LIN {X 0,Y 353.68,Z 667.866,A -85,B 0,C 180,E1 -13495.441,E2 -13495.441} C_VEL
LIN {X 0,Y 353.682,Z 668.66,A -85,B 0,C 180,E1 -13496.583,E2 -13496.583} C_VEL
LIN {X 0,Y 353.463,Z 669.191,A -85,B 0,C 180,E1 -13498.861,E2 -13498.861} C_VEL
LIN {X 0,Y 353.397,Z 668.253,A -85,B 0,C 180,E1 -13501.14,E2 -13501.14} C_VEL
LIN {X 0,Y 353.398,Z 665.846,A -85,B 0,C 180,E1 -13503.42,E2 -13503.42} C_VEL
LIN {X 0,Y 353.541,Z 663.076,A -85,B 0,C 180,E1 -13505.132,E2 -13505.132} C_VEL
LIN {X 0,Y 353.829,Z 657.939,A -85,B 0,C 180,E1 -13507.418,E2 -13507.418} C_VEL
LIN {X 0,Y 354.1,Z 652.954,A -85,B 0,C 180,E1 -13509.136,E2 -13509.136} C_VEL
LIN {X 0,Y 354.652,Z 645.736,A -85,B 0,C 180,E1 -13511.14,E2 -13511.14} C_VEL
LIN {X 0,Y 355.365,Z 638.179,A -85,B 0,C 180,E1 -13512.855,E2 -13512.855} C_VEL
LIN {X 0,Y 356.178,Z 628.788,A -85,B 0,C 180,E1 -13514.626,E2 -13514.626} C_VEL
LIN {X 0,Y 357.149,Z 618.14,A -85,B 0,C 180,E1 -13516.285,E2 -13516.285} C_VEL
LIN {X 0,Y 358.299,Z 605.968,A -85,B 0,C 180,E1 -13517.848,E2 -13517.848} C_VEL
LIN {X 0,Y 359.381,Z 593.917,A -85,B 0,C 180,E1 -13519.121,E2 -13519.121} C_VEL
LIN {X 0,Y 360.455,Z 580.861,A -85,B 0,C 180,E1 -13520.248,E2 -13520.248} C_VEL
LIN {X 0,Y 361.486,Z 566.317,A -85,B 0,C 180,E1 -13521.237,E2 -13521.237} C_VEL
LIN {X 0,Y 362.333,Z 551.357,A -85,B 0,C 180,E1 -13521.999,E2 -13521.999} C_VEL
LIN {X 0,Y 363.06,Z 535.678,A -85,B 0,C 180,E1 -13522.552,E2 -13522.552} C_VEL
LIN {X 0,Y 366.741,Z 431.293,A -85,B 0,C 180,E1 -13525.312,E2 -13525.312} C_VEL
LIN {X 0,Y 361.436,Z 398.032,A -85,B 0,C 180,E1 -13526.613,E2 -13526.613} C_VEL
LIN {X 0,Y 361.949,Z 391.941,A -85,B 0,C 180,E1 -13527.776,E2 -13527.776} C_VEL
LIN {X 0,Y 359.699,Z 381.366,A -85,B 0,C 180,E1 -13530.108,E2 -13530.108} C_VEL
LIN {X 0,Y 356.197,Z 366.492,A -85,B 0,C 180,E1 -13533.536,E2 -13533.536} C_VEL
LIN {X 0,Y 354.88,Z 361.062,A -85,B 0,C 180,E1 -13534.895,E2 -13534.895} C_VEL
LIN {X 0,Y 354.793,Z 360.917,A -85,B 0,C 180,E1 -13537.885,E2 -13537.885} C_VEL
LIN {X 0,Y 354.768,Z 360.912,A -85,B 0,C 180,E1 -13541.167,E2 -13541.167} C_VEL
LIN {X 0,Y 354.759,Z 360.919,A -85,B 0,C 180,E1 -13544.505,E2 -13544.505} C_VEL
LIN {X 0,Y 354.782,Z 360.903,A -85,B 0,C 180,E1 -13547.661,E2 -13547.661} C_VEL
LIN {X 0,Y 354.804,Z 361.09,A -85,B 0,C 180,E1 -13551.115,E2 -13551.115} C_VEL
LIN {X 0,Y 359.178,Z 374.687,A -85,B 0,C 180,E1 -13554.055,E2 -13554.055} C_VEL
LIN {X 0,Y 363.071,Z 388.801,A -85,B 0,C 180,E1 -13556.835,E2 -13556.835} C_VEL
LIN {X 0,Y 365.06,Z 396.769,A -85,B 0,C 180,E1 -13558.239,E2 -13558.239} C_VEL
LIN {X 0,Y 367.606,Z 402.868,A -85,B 0,C 180,E1 -13558.628,E2 -13558.628} C_VEL
LIN {X 0,Y 372.329,Z 427.279,A -85,B 0,C 180,E1 -13559.605,E2 -13559.605} C_VEL
LIN {X 0,Y 373.954,Z 436.927,A -85,B 0,C 180,E1 -13559.961,E2 -13559.961} C_VEL
LIN {X 0,Y 370.986,Z 551.693,A -85,B 0,C 180,E1 -13562.193,E2 -13562.193} C_VEL
LIN {X 0,Y 370.367,Z 569.388,A -85,B 0,C 180,E1 -13562.602,E2 -13562.602} C_VEL
LIN {X 0,Y 369.3,Z 584.628,A -85,B 0,C 180,E1 -13563.16,E2 -13563.16} C_VEL
LIN {X 0,Y 368.135,Z 598.529,A -85,B 0,C 180,E1 -13563.879,E2 -13563.879} C_VEL
LIN {X 0,Y 366.76,Z 611.782,A -85,B 0,C 180,E1 -13564.764,E2 -13564.764} C_VEL
LIN {X 0,Y 365.042,Z 624.849,A -85,B 0,C 180,E1 -13565.85,E2 -13565.85} C_VEL
LIN {X 0,Y 363.164,Z 638.241,A -85,B 0,C 180,E1 -13567.229,E2 -13567.229} C_VEL
LIN {X 0,Y 361.199,Z 650.71,A -85,B 0,C 180,E1 -13568.797,E2 -13568.797} C_VEL
LIN {X 0,Y 359.445,Z 662.34,A -85,B 0,C 180,E1 -13570.586,E2 -13570.586} C_VEL
LIN {X 0,Y 357.872,Z 671.556,A -85,B 0,C 180,E1 -13572.278,E2 -13572.278} C_VEL
LIN {X 0,Y 356.387,Z 680.618,A -85,B 0,C 180,E1 -13574.267,E2 -13574.267} C_VEL
LIN {X 0,Y 355.315,Z 688.145,A -85,B 0,C 180,E1 -13576.269,E2 -13576.269} C_VEL
LIN {X 0,Y 354.332,Z 695.165,A -85,B 0,C 180,E1 -13578.56,E2 -13578.56} C_VEL
LIN {X 0,Y 353.76,Z 700.689,A -85,B 0,C 180,E1 -13580.855,E2 -13580.855} C_VEL
LIN {X 0,Y 353.349,Z 704.87,A -85,B 0,C 180,E1 -13583.146,E2 -13583.146} C_VEL
LIN {X 0,Y 353.251,Z 706.641,A -85,B 0,C 180,E1 -13584.422,E2 -13584.422} C_VEL
LIN {X 0,Y 352.529,Z 707.753,A -85,B 0,C 180,E1 -13585.359,E2 -13585.359} C_VEL
LIN {X 0,Y 349.602,Z 709.065,A -85,B 0,C 180,E1 -13586.891,E2 -13586.891} C_VEL
LIN {X 0,Y 347.154,Z 709.751,A -85,B 0,C 180,E1 -13588.137,E2 -13588.137} C_VEL
LIN {X 0,Y 346.11,Z 710.054,A -85,B 0,C 180,E1 -13589.105,E2 -13589.105} C_VEL
LIN {X 0,Y 346.028,Z 710.09,A -85,B 0,C 180,E1 -13589.433,E2 -13589.433} C_VEL
LIN {X 0,Y 346.047,Z 710.023,A -85,B 0,C 180,E1 -13591.164,E2 -13591.164} C_VEL
LIN {X 0,Y 346.111,Z 708.885,A -85,B 0,C 180,E1 -13593.492,E2 -13593.492} C_VEL
LIN {X 0,Y 346.234,Z 706.453,A -85,B 0,C 180,E1 -13595.943,E2 -13595.943} C_VEL
LIN {X 0,Y 346.495,Z 703.113,A -85,B 0,C 180,E1 -13598.162,E2 -13598.162} C_VEL
LIN {X 0,Y 346.944,Z 698.339,A -85,B 0,C 180,E1 -13600.504,E2 -13600.504} C_VEL
LIN {X 0,Y 347.846,Z 692.148,A -85,B 0,C 180,E1 -13602.841,E2 -13602.841} C_VEL
LIN {X 0,Y 348.924,Z 684.367,A -85,B 0,C 180,E1 -13605.179,E2 -13605.179} C_VEL
LIN {X 0,Y 350.291,Z 676.075,A -85,B 0,C 180,E1 -13607.213,E2 -13607.213} C_VEL
LIN {X 0,Y 352.021,Z 666.081,A -85,B 0,C 180,E1 -13609.233,E2 -13609.233} C_VEL
LIN {X 0,Y 353.694,Z 655.876,A -85,B 0,C 180,E1 -13610.957,E2 -13610.957} C_VEL
LIN {X 0,Y 355.739,Z 643.656,A -85,B 0,C 180,E1 -13612.659,E2 -13612.659} C_VEL
LIN {X 0,Y 357.622,Z 631.43,A -85,B 0,C 180,E1 -13614.065,E2 -13614.065} C_VEL
LIN {X 0,Y 359.524,Z 618.079,A -85,B 0,C 180,E1 -13615.316,E2 -13615.316} C_VEL
LIN {X 0,Y 361.249,Z 603.581,A -85,B 0,C 180,E1 -13616.401,E2 -13616.401} C_VEL
LIN {X 0,Y 362.608,Z 588.97,A -85,B 0,C 180,E1 -13617.247,E2 -13617.247} C_VEL
LIN {X 0,Y 363.79,Z 574.332,A -85,B 0,C 180,E1 -13617.857,E2 -13617.857} C_VEL
LIN {X 0,Y 364.615,Z 558.128,A -85,B 0,C 180,E1 -13618.297,E2 -13618.297} C_VEL
LIN {X 0,Y 367.783,Z 437.247,A -85,B 0,C 180,E1 -13620.693,E2 -13620.693} C_VEL
LIN {X 0,Y 362.784,Z 410.112,A -85,B 0,C 180,E1 -13621.778,E2 -13621.778} C_VEL
LIN {X 0,Y 361.54,Z 404.727,A -85,B 0,C 180,E1 -13622.023,E2 -13622.023} C_VEL
LIN {X 0,Y 357.822,Z 396.238,A -85,B 0,C 180,E1 -13622.622,E2 -13622.622} C_VEL
LIN {X 0,Y 354.484,Z 383.285,A -85,B 0,C 180,E1 -13625.096,E2 -13625.096} C_VEL
LIN {X 0,Y 350.708,Z 370.946,A -85,B 0,C 180,E1 -13627.668,E2 -13627.668} C_VEL
LIN {X 0,Y 347.74,Z 361.921,A -85,B 0,C 180,E1 -13629.736,E2 -13629.736} C_VEL
LIN {X 0,Y 347.722,Z 361.796,A -85,B 0,C 180,E1 -13633.408,E2 -13633.408} C_VEL
LIN {X 0,Y 347.724,Z 361.799,A -85,B 0,C 180,E1 -13636.686,E2 -13636.686} C_VEL
LIN {X 0,Y 347.701,Z 361.796,A -85,B 0,C 180,E1 -13640.182,E2 -13640.182} C_VEL
LIN {X 0,Y 347.754,Z 361.793,A -85,B 0,C 180,E1 -13642.678,E2 -13642.678} C_VEL
LIN {X 0,Y 347.748,Z 361.793,A -85,B 0,C 180,E1 -13645.956,E2 -13645.956} C_VEL
LIN {X 0,Y 347.738,Z 361.789,A -85,B 0,C 180,E1 -13649.651,E2 -13649.651} C_VEL
LIN {X 0,Y 347.748,Z 361.78,A -85,B 0,C 180,E1 -13653.601,E2 -13653.601} C_VEL
LIN {X 0,Y 347.756,Z 361.787,A -85,B 0,C 180,E1 -13656.159,E2 -13656.159} C_VEL
LIN {X 0,Y 347.8,Z 361.787,A -85,B 0,C 180,E1 -13659.908,E2 -13659.908} C_VEL
LIN {X 0,Y 347.832,Z 361.765,A -85,B 0,C 180,E1 -13663.568,E2 -13663.568} C_VEL
LIN {X 0,Y 347.89,Z 361.772,A -85,B 0,C 180,E1 -13667.16,E2 -13667.16} C_VEL
LIN {X 0,Y 347.936,Z 361.762,A -85,B 0,C 180,E1 -13670.7,E2 -13670.7} C_VEL
LIN {X 0,Y 348.079,Z 361.75,A -85,B 0,C 180,E1 -13673.042,E2 -13673.042} C_VEL
LIN {X 0,Y 348.195,Z 361.737,A -85,B 0,C 180,E1 -13677.686,E2 -13677.686} C_VEL
LIN {X 0,Y 348.324,Z 361.711,A -85,B 0,C 180,E1 -13680,E2 -13680} C_VEL
LIN {X 0,Y 348.204,Z 361.719,A -85,B 0,C 180,E1 -13682.313,E2 -13682.313} C_VEL
LIN {X 0,Y 348.068,Z 361.735,A -85,B 0,C 180,E1 -13686.958,E2 -13686.958} C_VEL
LIN {X 0,Y 347.897,Z 361.771,A -85,B 0,C 180,E1 -13690.475,E2 -13690.475} C_VEL
LIN {X 0,Y 347.899,Z 361.753,A -85,B 0,C 180,E1 -13694.15,E2 -13694.15} C_VEL
LIN {X 0,Y 347.829,Z 361.776,A -85,B 0,C 180,E1 -13698.259,E2 -13698.259} C_VEL
LIN {X 0,Y 347.79,Z 361.787,A -85,B 0,C 180,E1 -13701.636,E2 -13701.636} C_VEL
LIN {X 0,Y 347.812,Z 361.769,A -85,B 0,C 180,E1 -13705.108,E2 -13705.108} C_VEL
LIN {X 0,Y 347.811,Z 361.785,A -85,B 0,C 180,E1 -13707.694,E2 -13707.694} C_VEL
LIN {X 0,Y 347.764,Z 361.777,A -85,B 0,C 180,E1 -13710.346,E2 -13710.346} C_VEL
LIN {X 0,Y 347.744,Z 361.781,A -85,B 0,C 180,E1 -13714.464,E2 -13714.464} C_VEL
LIN {X 0,Y 347.772,Z 361.774,A -85,B 0,C 180,E1 -13717.988,E2 -13717.988} C_VEL
LIN {X 0,Y 347.75,Z 361.762,A -85,B 0,C 180,E1 -13721.83,E2 -13721.83} C_VEL
LIN {X 0,Y 347.706,Z 361.782,A -85,B 0,C 180,E1 -13725.027,E2 -13725.027} C_VEL
LIN {X 0,Y 347.75,Z 361.775,A -85,B 0,C 180,E1 -13728.397,E2 -13728.397} C_VEL
LIN {X 0,Y 347.8,Z 362.002,A -85,B 0,C 180,E1 -13732.115,E2 -13732.115} C_VEL
LIN {X 0,Y 351.917,Z 377.162,A -85,B 0,C 180,E1 -13735.434,E2 -13735.434} C_VEL
LIN {X 0,Y 353.136,Z 382.059,A -85,B 0,C 180,E1 -13736.431,E2 -13736.431} C_VEL
LIN {X 0,Y 356.826,Z 392.05,A -85,B 0,C 180,E1 -13737.524,E2 -13737.524} C_VEL
LIN {X 0,Y 362.533,Z 405.129,A -85,B 0,C 180,E1 -13738.398,E2 -13738.398} C_VEL
LIN {X 0,Y 367.206,Z 434.33,A -85,B 0,C 180,E1 -13739.498,E2 -13739.498} C_VEL
LIN {X 0,Y 363.912,Z 560.453,A -85,B 0,C 180,E1 -13741.996,E2 -13741.996} C_VEL
LIN {X 0,Y 363.111,Z 575.693,A -85,B 0,C 180,E1 -13742.438,E2 -13742.438} C_VEL
LIN {X 0,Y 361.972,Z 590.5,A -85,B 0,C 180,E1 -13743.087,E2 -13743.087} C_VEL
LIN {X 0,Y 360.774,Z 603.077,A -85,B 0,C 180,E1 -13743.822,E2 -13743.822} C_VEL
LIN {X 0,Y 359.191,Z 616.425,A -85,B 0,C 180,E1 -13744.814,E2 -13744.814} C_VEL
LIN {X 0,Y 357.269,Z 629.979,A -85,B 0,C 180,E1 -13746.064,E2 -13746.064} C_VEL
LIN {X 0,Y 355.271,Z 643.469,A -85,B 0,C 180,E1 -13747.617,E2 -13747.617} C_VEL
LIN {X 0,Y 353.499,Z 654.325,A -85,B 0,C 180,E1 -13749.134,E2 -13749.134} C_VEL
LIN {X 0,Y 351.659,Z 665.693,A -85,B 0,C 180,E1 -13751.049,E2 -13751.049} C_VEL
LIN {X 0,Y 349.986,Z 675.576,A -85,B 0,C 180,E1 -13753.072,E2 -13753.072} C_VEL
LIN {X 0,Y 348.605,Z 684.331,A -85,B 0,C 180,E1 -13755.262,E2 -13755.262} C_VEL
LIN {X 0,Y 347.529,Z 692.258,A -85,B 0,C 180,E1 -13757.741,E2 -13757.741} C_VEL
LIN {X 0,Y 346.802,Z 698.165,A -85,B 0,C 180,E1 -13760.081,E2 -13760.081} C_VEL
LIN {X 0,Y 346.48,Z 701.649,A -85,B 0,C 180,E1 -13761.837,E2 -13761.837} C_VEL
LIN {X 0,Y 346.199,Z 705.184,A -85,B 0,C 180,E1 -13764.174,E2 -13764.174} C_VEL
LIN {X 0,Y 346.128,Z 707.51,A -85,B 0,C 180,E1 -13766.508,E2 -13766.508} C_VEL
LIN {X 0,Y 346.059,Z 708.68,A -85,B 0,C 180,E1 -13768.836,E2 -13768.836} C_VEL
LIN {X 0,Y 346.06,Z 708.679,A -85,B 0,C 180,E1 -13771.164,E2 -13771.164} C_VEL
LIN {X 0,Y 346.13,Z 707.506,A -85,B 0,C 180,E1 -13773.492,E2 -13773.492} C_VEL
LIN {X 0,Y 346.232,Z 705.027,A -85,B 0,C 180,E1 -13775.944,E2 -13775.944} C_VEL
LIN {X 0,Y 346.593,Z 700.563,A -85,B 0,C 180,E1 -13778.748,E2 -13778.748} C_VEL
LIN {X 0,Y 347.072,Z 695.361,A -85,B 0,C 180,E1 -13781.091,E2 -13781.091} C_VEL
LIN {X 0,Y 347.981,Z 688.704,A -85,B 0,C 180,E1 -13783.43,E2 -13783.43} C_VEL
LIN {X 0,Y 349.228,Z 680.389,A -85,B 0,C 180,E1 -13785.764,E2 -13785.764} C_VEL
LIN {X 0,Y 350.666,Z 671.482,A -85,B 0,C 180,E1 -13787.797,E2 -13787.797} C_VEL
LIN {X 0,Y 352.22,Z 662.383,A -85,B 0,C 180,E1 -13789.525,E2 -13789.525} C_VEL
LIN {X 0,Y 353.964,Z 651.632,A -85,B 0,C 180,E1 -13791.245,E2 -13791.245} C_VEL
LIN {X 0,Y 355.82,Z 639.874,A -85,B 0,C 180,E1 -13792.807,E2 -13792.807} C_VEL
LIN {X 0,Y 357.728,Z 627.004,A -85,B 0,C 180,E1 -13794.212,E2 -13794.212} C_VEL
LIN {X 0,Y 359.429,Z 614.507,A -85,B 0,C 180,E1 -13795.324,E2 -13795.324} C_VEL
LIN {X 0,Y 362.493,Z 591.653,A -85,B 0,C 180,E1 -13797.019,E2 -13797.019} C_VEL
LIN {X 0,Y 364.417,Z 576.794,A -85,B 0,C 180,E1 -13797.884,E2 -13797.884} C_VEL
LIN {X 0,Y 366.213,Z 560.409,A -85,B 0,C 180,E1 -13798.593,E2 -13798.593} C_VEL
LIN {X 0,Y 373.017,Z 477.293,A -85,B 0,C 180,E1 -13801.167,E2 -13801.167} C_VEL
LIN {X 0,Y 376.881,Z 436.762,A -85,B 0,C 180,E1 -13802.478,E2 -13802.478} C_VEL
LIN {X 0,Y 375.821,Z 423.937,A -85,B 0,C 180,E1 -13803.36,E2 -13803.36} C_VEL
LIN {X 0,Y 375.337,Z 421.498,A -85,B 0,C 180,E1 -13803.594,E2 -13803.594} C_VEL
LIN {X 0,Y 372.439,Z 415.253,A -85,B 0,C 180,E1 -13804.586,E2 -13804.586} C_VEL
LIN {X 0,Y 369.189,Z 409.492,A -85,B 0,C 180,E1 -13805.762,E2 -13805.762} C_VEL
LIN {X 0,Y 366.165,Z 404.402,A -85,B 0,C 180,E1 -13807.009,E2 -13807.009} C_VEL
LIN {X 0,Y 363.079,Z 399.436,A -85,B 0,C 180,E1 -13808.569,E2 -13808.569} C_VEL
LIN {X 0,Y 362.44,Z 397.459,A -85,B 0,C 180,E1 -13809.784,E2 -13809.784} C_VEL
LIN {X 0,Y 361.471,Z 394.656,A -85,B 0,C 180,E1 -13812.369,E2 -13812.369} C_VEL
LIN {X 0,Y 361.043,Z 393.422,A -85,B 0,C 180,E1 -13814.489,E2 -13814.489} C_VEL
LIN {X 0,Y 360.859,Z 393.255,A -85,B 0,C 180,E1 -13817.027,E2 -13817.027} C_VEL
LIN {X 0,Y 361.126,Z 394.24,A -85,B 0,C 180,E1 -13819.376,E2 -13819.376} C_VEL
LIN {X 0,Y 361.654,Z 396.163,A -85,B 0,C 180,E1 -13821.548,E2 -13821.548} C_VEL
LIN {X 0,Y 362.499,Z 399.525,A -85,B 0,C 180,E1 -13823.9,E2 -13823.9} C_VEL
LIN {X 0,Y 366.576,Z 406.402,A -85,B 0,C 180,E1 -13825.972,E2 -13825.972} C_VEL
LIN {X 0,Y 369.665,Z 412.043,A -85,B 0,C 180,E1 -13827.267,E2 -13827.267} C_VEL
LIN {X 0,Y 372.445,Z 417.629,A -85,B 0,C 180,E1 -13828.32,E2 -13828.32} C_VEL
LIN {X 0,Y 373.974,Z 421.159,A -85,B 0,C 180,E1 -13828.882,E2 -13828.882} C_VEL
LIN {X 0,Y 375.802,Z 433.348,A -85,B 0,C 180,E1 -13829.979,E2 -13829.979} C_VEL
LIN {X 0,Y 376.409,Z 439.645,A -85,B 0,C 180,E1 -13830.448,E2 -13830.448} C_VEL
LIN {X 0,Y 367.997,Z 523.078,A -85,B 0,C 180,E1 -13833.333,E2 -13833.333} C_VEL
LIN {X 0,Y 365.648,Z 549.794,A -85,B 0,C 180,E1 -13834.3,E2 -13834.3} C_VEL
LIN {X 0,Y 363.925,Z 565.425,A -85,B 0,C 180,E1 -13835.101,E2 -13835.101} C_VEL
LIN {X 0,Y 361.927,Z 580.859,A -85,B 0,C 180,E1 -13836.168,E2 -13836.168} C_VEL
LIN {X 0,Y 359.954,Z 594.107,A -85,B 0,C 180,E1 -13837.318,E2 -13837.318} C_VEL
LIN {X 0,Y 357.813,Z 607.057,A -85,B 0,C 180,E1 -13838.693,E2 -13838.693} C_VEL
LIN {X 0,Y 356.004,Z 617.795,A -85,B 0,C 180,E1 -13840.09,E2 -13840.09} C_VEL
LIN {X 0,Y 354.091,Z 628.587,A -85,B 0,C 180,E1 -13841.784,E2 -13841.784} C_VEL
LIN {X 0,Y 352.259,Z 637.817,A -85,B 0,C 180,E1 -13843.517,E2 -13843.517} C_VEL
LIN {X 0,Y 350.647,Z 646.382,A -85,B 0,C 180,E1 -13845.491,E2 -13845.491} C_VEL
LIN {X 0,Y 349.487,Z 652.555,A -85,B 0,C 180,E1 -13847.22,E2 -13847.22} C_VEL
LIN {X 0,Y 348.612,Z 657.656,A -85,B 0,C 180,E1 -13848.959,E2 -13848.959} C_VEL
LIN {X 0,Y 347.849,Z 661.742,A -85,B 0,C 180,E1 -13850.698,E2 -13850.698} C_VEL
LIN {X 0,Y 347.137,Z 665.827,A -85,B 0,C 180,E1 -13853.023,E2 -13853.023} C_VEL
LIN {X 0,Y 346.615,Z 668.423,A -85,B 0,C 180,E1 -13855.348,E2 -13855.348} C_VEL
LIN {X 0,Y 346.599,Z 669.156,A -85,B 0,C 180,E1 -13856.513,E2 -13856.513} C_VEL
LIN {X 0,Y 346.514,Z 669.535,A -85,B 0,C 180,E1 -13857.675,E2 -13857.675} C_VEL
LIN {X 0,Y 346.324,Z 669.205,A -85,B 0,C 180,E1 -13860,E2 -13860} C_VEL
LIN {X 0,Y 346.301,Z 667.422,A -85,B 0,C 180,E1 -13862.326,E2 -13862.326} C_VEL
LIN {X 0,Y 346.417,Z 664.153,A -85,B 0,C 180,E1 -13864.655,E2 -13864.655} C_VEL
LIN {X 0,Y 346.7,Z 659.314,A -85,B 0,C 180,E1 -13866.986,E2 -13866.986} C_VEL
LIN {X 0,Y 346.912,Z 654.543,A -85,B 0,C 180,E1 -13868.74,E2 -13868.74} C_VEL
LIN {X 0,Y 347.482,Z 647.628,A -85,B 0,C 180,E1 -13870.783,E2 -13870.783} C_VEL
LIN {X 0,Y 348.242,Z 639.047,A -85,B 0,C 180,E1 -13872.826,E2 -13872.826} C_VEL
LIN {X 0,Y 349.145,Z 628.988,A -85,B 0,C 180,E1 -13874.77,E2 -13874.77} C_VEL
LIN {X 0,Y 350.163,Z 618.248,A -85,B 0,C 180,E1 -13876.469,E2 -13876.469} C_VEL
LIN {X 0,Y 351.336,Z 606.022,A -85,B 0,C 180,E1 -13878.063,E2 -13878.063} C_VEL
LIN {X 0,Y 352.447,Z 593.918,A -85,B 0,C 180,E1 -13879.361,E2 -13879.361} C_VEL
LIN {X 0,Y 353.569,Z 580.812,A -85,B 0,C 180,E1 -13880.508,E2 -13880.508} C_VEL
LIN {X 0,Y 354.557,Z 567.451,A -85,B 0,C 180,E1 -13881.441,E2 -13881.441} C_VEL
LIN {X 0,Y 355.438,Z 551.999,A -85,B 0,C 180,E1 -13882.258,E2 -13882.258} C_VEL
LIN {X 0,Y 356.191,Z 536.686,A -85,B 0,C 180,E1 -13882.82,E2 -13882.82} C_VEL
LIN {X 0,Y 360.063,Z 432.773,A -85,B 0,C 180,E1 -13885.652,E2 -13885.652} C_VEL
LIN {X 0,Y 354.636,Z 397.9,A -85,B 0,C 180,E1 -13887.045,E2 -13887.045} C_VEL
LIN {X 0,Y 354.997,Z 392.861,A -85,B 0,C 180,E1 -13888.047,E2 -13888.047} C_VEL
LIN {X 0,Y 352.187,Z 380.215,A -85,B 0,C 180,E1 -13890.898,E2 -13890.898} C_VEL
LIN {X 0,Y 348.718,Z 365.637,A -85,B 0,C 180,E1 -13894.354,E2 -13894.354} C_VEL
LIN {X 0,Y 347.852,Z 362.086,A -85,B 0,C 180,E1 -13895.245,E2 -13895.245} C_VEL
LIN {X 0,Y 347.785,Z 361.79,A -85,B 0,C 180,E1 -13895.876,E2 -13895.876} C_VEL
LIN {X 0,Y 347.731,Z 361.796,A -85,B 0,C 180,E1 -13898.796,E2 -13898.796} C_VEL
LIN {X 0,Y 347.74,Z 361.776,A -85,B 0,C 180,E1 -13901.832,E2 -13901.832} C_VEL
LIN {X 0,Y 347.701,Z 361.801,A -85,B 0,C 180,E1 -13905.028,E2 -13905.028} C_VEL
LIN {X 0,Y 347.738,Z 361.79,A -85,B 0,C 180,E1 -13908.4,E2 -13908.4} C_VEL
LIN {X 0,Y 347.756,Z 362.047,A -85,B 0,C 180,E1 -13910.443,E2 -13910.443} C_VEL
LIN {X 0,Y 352.21,Z 375.538,A -85,B 0,C 180,E1 -13913.431,E2 -13913.431} C_VEL
LIN {X 0,Y 355.861,Z 388.48,A -85,B 0,C 180,E1 -13916.045,E2 -13916.045} C_VEL
LIN {X 0,Y 357.939,Z 396.68,A -85,B 0,C 180,E1 -13917.531,E2 -13917.531} C_VEL
LIN {X 0,Y 361.828,Z 405.67,A -85,B 0,C 180,E1 -13918.135,E2 -13918.135} C_VEL
LIN {X 0,Y 366.446,Z 430.021,A -85,B 0,C 180,E1 -13919.128,E2 -13919.128} C_VEL
LIN {X 0,Y 367.786,Z 437.374,A -85,B 0,C 180,E1 -13919.416,E2 -13919.416} C_VEL
LIN {X 0,Y 364.86,Z 548.023,A -85,B 0,C 180,E1 -13921.606,E2 -13921.606} C_VEL
LIN {X 0,Y 364.166,Z 568.265,A -85,B 0,C 180,E1 -13922.056,E2 -13922.056} C_VEL
LIN {X 0,Y 363.068,Z 583.786,A -85,B 0,C 180,E1 -13922.618,E2 -13922.618} C_VEL
LIN {X 0,Y 361.786,Z 598.297,A -85,B 0,C 180,E1 -13923.371,E2 -13923.371} C_VEL
LIN {X 0,Y 360.315,Z 611.947,A -85,B 0,C 180,E1 -13924.296,E2 -13924.296} C_VEL
LIN {X 0,Y 358.563,Z 624.825,A -85,B 0,C 180,E1 -13925.385,E2 -13925.385} C_VEL
LIN {X 0,Y 356.595,Z 638.22,A -85,B 0,C 180,E1 -13926.785,E2 -13926.785} C_VEL
LIN {X 0,Y 354.553,Z 650.692,A -85,B 0,C 180,E1 -13928.38,E2 -13928.38} C_VEL
LIN {X 0,Y 352.713,Z 662.323,A -85,B 0,C 180,E1 -13930.2,E2 -13930.2} C_VEL
LIN {X 0,Y 351.073,Z 671.54,A -85,B 0,C 180,E1 -13931.923,E2 -13931.923} C_VEL
LIN {X 0,Y 349.481,Z 680.603,A -85,B 0,C 180,E1 -13933.948,E2 -13933.948} C_VEL
LIN {X 0,Y 348.366,Z 688.13,A -85,B 0,C 180,E1 -13935.99,E2 -13935.99} C_VEL
LIN {X 0,Y 347.342,Z 695.152,A -85,B 0,C 180,E1 -13938.326,E2 -13938.326} C_VEL
LIN {X 0,Y 346.705,Z 700.676,A -85,B 0,C 180,E1 -13940.667,E2 -13940.667} C_VEL
LIN {X 0,Y 346.29,Z 704.857,A -85,B 0,C 180,E1 -13943.006,E2 -13943.006} C_VEL
LIN {X 0,Y 346.132,Z 707.795,A -85,B 0,C 180,E1 -13945.341,E2 -13945.341} C_VEL
LIN {X 0,Y 346.043,Z 709.556,A -85,B 0,C 180,E1 -13947.672,E2 -13947.672} C_VEL
LIN {X 0,Y 346.028,Z 710.09,A -85,B 0,C 180,E1 -13949.433,E2 -13949.433} C_VEL
LIN {X 0,Y 345.362,Z 710.139,A -85,B 0,C 180,E1 -13950.404,E2 -13950.404} C_VEL
LIN {X 0,Y 342.505,Z 709.738,A -85,B 0,C 180,E1 -13951.984,E2 -13951.984} C_VEL
LIN {X 0,Y 340.103,Z 709.07,A -85,B 0,C 180,E1 -13953.259,E2 -13953.259} C_VEL
LIN {X 0,Y 339.1,Z 708.353,A -85,B 0,C 180,E1 -13954.242,E2 -13954.242} C_VEL
LIN {X 0,Y 339.034,Z 708.025,A -85,B 0,C 180,E1 -13954.575,E2 -13954.575} C_VEL
LIN {X 0,Y 339.252,Z 704.995,A -85,B 0,C 180,E1 -13957.14,E2 -13957.14} C_VEL
LIN {X 0,Y 339.648,Z 700.878,A -85,B 0,C 180,E1 -13959.528,E2 -13959.528} C_VEL
LIN {X 0,Y 340.337,Z 695.413,A -85,B 0,C 180,E1 -13961.917,E2 -13961.917} C_VEL
LIN {X 0,Y 341.373,Z 688.452,A -85,B 0,C 180,E1 -13964.303,E2 -13964.303} C_VEL
LIN {X 0,Y 342.792,Z 679.786,A -85,B 0,C 180,E1 -13966.68,E2 -13966.68} C_VEL
LIN {X 0,Y 344.419,Z 670.56,A -85,B 0,C 180,E1 -13968.747,E2 -13968.747} C_VEL
LIN {X 0,Y 346.329,Z 660.206,A -85,B 0,C 180,E1 -13970.662,E2 -13970.662} C_VEL
LIN {X 0,Y 348.222,Z 648.981,A -85,B 0,C 180,E1 -13972.392,E2 -13972.392} C_VEL
LIN {X 0,Y 350.336,Z 636.534,A -85,B 0,C 180,E1 -13973.968,E2 -13973.968} C_VEL
LIN {X 0,Y 352.207,Z 624.297,A -85,B 0,C 180,E1 -13975.247,E2 -13975.247} C_VEL
LIN {X 0,Y 354.079,Z 610.676,A -85,B 0,C 180,E1 -13976.4,E2 -13976.4} C_VEL
LIN {X 0,Y 355.643,Z 596.521,A -85,B 0,C 180,E1 -13977.352,E2 -13977.352} C_VEL
LIN {X 0,Y 356.83,Z 583.747,A -85,B 0,C 180,E1 -13978.009,E2 -13978.009} C_VEL
LIN {X 0,Y 357.895,Z 568.931,A -85,B 0,C 180,E1 -13978.557,E2 -13978.557} C_VEL
LIN {X 0,Y 358.588,Z 550.914,A -85,B 0,C 180,E1 -13978.977,E2 -13978.977} C_VEL
LIN {X 0,Y 361.68,Z 438.308,A -85,B 0,C 180,E1 -13981.241,E2 -13981.241} C_VEL
LIN {X 0,Y 356.144,Z 408.487,A -85,B 0,C 180,E1 -13982.476,E2 -13982.476} C_VEL
LIN {X 0,Y 350.747,Z 396.094,A -85,B 0,C 180,E1 -13983.371,E2 -13983.371} C_VEL
LIN {X 0,Y 346.906,Z 381.93,A -85,B 0,C 180,E1 -13986.18,E2 -13986.18} C_VEL
LIN {X 0,Y 342.944,Z 369.556,A -85,B 0,C 180,E1 -13988.855,E2 -13988.855} C_VEL
LIN {X 0,Y 340.701,Z 362.896,A -85,B 0,C 180,E1 -13990.432,E2 -13990.432} C_VEL
LIN {X 0,Y 340.693,Z 362.67,A -85,B 0,C 180,E1 -13992.044,E2 -13992.044} C_VEL
LIN {X 0,Y 340.651,Z 362.681,A -85,B 0,C 180,E1 -13996.227,E2 -13996.227} C_VEL
LIN {X 0,Y 340.671,Z 362.675,A -85,B 0,C 180,E1 -13998.688,E2 -13998.688} C_VEL
LIN {X 0,Y 340.718,Z 362.664,A -85,B 0,C 180,E1 -14001.77,E2 -14001.77} C_VEL
LIN {X 0,Y 340.722,Z 362.663,A -85,B 0,C 180,E1 -14005.596,E2 -14005.596} C_VEL
LIN {X 0,Y 340.693,Z 362.66,A -85,B 0,C 180,E1 -14008.955,E2 -14008.955} C_VEL
LIN {X 0,Y 340.72,Z 362.652,A -85,B 0,C 180,E1 -14013.013,E2 -14013.013} C_VEL
LIN {X 0,Y 340.744,Z 362.666,A -85,B 0,C 180,E1 -14015.637,E2 -14015.637} C_VEL
LIN {X 0,Y 340.73,Z 362.661,A -85,B 0,C 180,E1 -14019.473,E2 -14019.473} C_VEL
LIN {X 0,Y 340.793,Z 362.648,A -85,B 0,C 180,E1 -14021.981,E2 -14021.981} C_VEL
LIN {X 0,Y 340.87,Z 362.651,A -85,B 0,C 180,E1 -14025.705,E2 -14025.705} C_VEL
LIN {X 0,Y 340.848,Z 362.632,A -85,B 0,C 180,E1 -14029.305,E2 -14029.305} C_VEL
LIN {X 0,Y 341.047,Z 362.627,A -85,B 0,C 180,E1 -14032.897,E2 -14032.897} C_VEL
LIN {X 0,Y 341.157,Z 362.613,A -85,B 0,C 180,E1 -14037.639,E2 -14037.639} C_VEL
LIN {X 0,Y 341.275,Z 362.589,A -85,B 0,C 180,E1 -14040,E2 -14040} C_VEL
LIN {X 0,Y 341.166,Z 362.595,A -85,B 0,C 180,E1 -14042.361,E2 -14042.361} C_VEL
LIN {X 0,Y 341.016,Z 362.611,A -85,B 0,C 180,E1 -14047.103,E2 -14047.103} C_VEL
LIN {X 0,Y 340.849,Z 362.649,A -85,B 0,C 180,E1 -14050.694,E2 -14050.694} C_VEL
LIN {X 0,Y 340.863,Z 362.629,A -85,B 0,C 180,E1 -14054.325,E2 -14054.325} C_VEL
LIN {X 0,Y 340.786,Z 362.649,A -85,B 0,C 180,E1 -14058.44,E2 -14058.44} C_VEL
LIN {X 0,Y 340.754,Z 362.664,A -85,B 0,C 180,E1 -14061.857,E2 -14061.857} C_VEL
LIN {X 0,Y 340.773,Z 362.649,A -85,B 0,C 180,E1 -14065.664,E2 -14065.664} C_VEL
LIN {X 0,Y 340.741,Z 362.665,A -85,B 0,C 180,E1 -14068.319,E2 -14068.319} C_VEL
LIN {X 0,Y 340.704,Z 362.662,A -85,B 0,C 180,E1 -14071.044,E2 -14071.044} C_VEL
LIN {X 0,Y 340.717,Z 362.66,A -85,B 0,C 180,E1 -14075.279,E2 -14075.279} C_VEL
LIN {X 0,Y 340.708,Z 362.643,A -85,B 0,C 180,E1 -14078.386,E2 -14078.386} C_VEL
LIN {X 0,Y 340.698,Z 362.643,A -85,B 0,C 180,E1 -14082.045,E2 -14082.045} C_VEL
LIN {X 0,Y 340.651,Z 362.642,A -85,B 0,C 180,E1 -14086.227,E2 -14086.227} C_VEL
LIN {X 0,Y 340.688,Z 362.673,A -85,B 0,C 180,E1 -14089.753,E2 -14089.753} C_VEL
LIN {X 0,Y 340.74,Z 362.861,A -85,B 0,C 180,E1 -14091.638,E2 -14091.638} C_VEL
LIN {X 0,Y 345.236,Z 379.417,A -85,B 0,C 180,E1 -14095.324,E2 -14095.324} C_VEL
LIN {X 0,Y 349.785,Z 391.999,A -85,B 0,C 180,E1 -14096.781,E2 -14096.781} C_VEL
LIN {X 0,Y 356.648,Z 407.397,A -85,B 0,C 180,E1 -14097.864,E2 -14097.864} C_VEL
LIN {X 0,Y 361.132,Z 436.155,A -85,B 0,C 180,E1 -14098.967,E2 -14098.967} C_VEL
LIN {X 0,Y 357.54,Z 563.496,A -85,B 0,C 180,E1 -14101.532,E2 -14101.532} C_VEL
LIN {X 0,Y 356.635,Z 578.466,A -85,B 0,C 180,E1 -14102.014,E2 -14102.014} C_VEL
LIN {X 0,Y 355.399,Z 593.12,A -85,B 0,C 180,E1 -14102.708,E2 -14102.708} C_VEL
LIN {X 0,Y 353.933,Z 607.132,A -85,B 0,C 180,E1 -14103.6,E2 -14103.6} C_VEL
LIN {X 0,Y 352.097,Z 621.247,A -85,B 0,C 180,E1 -14104.745,E2 -14104.745} C_VEL
LIN {X 0,Y 350.182,Z 633.914,A -85,B 0,C 180,E1 -14106.021,E2 -14106.021} C_VEL
LIN {X 0,Y 348.121,Z 646.684,A -85,B 0,C 180,E1 -14107.601,E2 -14107.601} C_VEL
LIN {X 0,Y 346.173,Z 658.437,A -85,B 0,C 180,E1 -14109.38,E2 -14109.38} C_VEL
LIN {X 0,Y 344.342,Z 668.683,A -85,B 0,C 180,E1 -14111.249,E2 -14111.249} C_VEL
LIN {X 0,Y 342.724,Z 678.05,A -85,B 0,C 180,E1 -14113.316,E2 -14113.316} C_VEL
LIN {X 0,Y 341.463,Z 685.575,A -85,B 0,C 180,E1 -14115.319,E2 -14115.319} C_VEL
LIN {X 0,Y 340.535,Z 692.275,A -85,B 0,C 180,E1 -14117.485,E2 -14117.485} C_VEL
LIN {X 0,Y 339.747,Z 698.18,A -85,B 0,C 180,E1 -14119.873,E2 -14119.873} C_VEL
LIN {X 0,Y 339.42,Z 701.664,A -85,B 0,C 180,E1 -14121.666,E2 -14121.666} C_VEL
LIN {X 0,Y 339.125,Z 705.285,A -85,B 0,C 180,E1 -14124.124,E2 -14124.124} C_VEL
LIN {X 0,Y 339.052,Z 707.524,A -85,B 0,C 180,E1 -14126.435,E2 -14126.435} C_VEL
LIN {X 0,Y 338.965,Z 708.693,A -85,B 0,C 180,E1 -14128.812,E2 -14128.812} C_VEL
LIN {X 0,Y 338.966,Z 708.692,A -85,B 0,C 180,E1 -14131.188,E2 -14131.188} C_VEL
LIN {X 0,Y 339.053,Z 707.519,A -85,B 0,C 180,E1 -14133.565,E2 -14133.565} C_VEL
LIN {X 0,Y 339.132,Z 705.187,A -85,B 0,C 180,E1 -14135.948,E2 -14135.948} C_VEL
LIN {X 0,Y 339.42,Z 701.638,A -85,B 0,C 180,E1 -14138.334,E2 -14138.334} C_VEL
LIN {X 0,Y 339.88,Z 696.792,A -85,B 0,C 180,E1 -14140.726,E2 -14140.726} C_VEL
LIN {X 0,Y 340.792,Z 690.519,A -85,B 0,C 180,E1 -14143.112,E2 -14143.112} C_VEL
LIN {X 0,Y 341.953,Z 682.627,A -85,B 0,C 180,E1 -14145.497,E2 -14145.497} C_VEL
LIN {X 0,Y 343.378,Z 674.193,A -85,B 0,C 180,E1 -14147.571,E2 -14147.571} C_VEL
LIN {X 0,Y 344.874,Z 665.636,A -85,B 0,C 180,E1 -14149.339,E2 -14149.339} C_VEL
LIN {X 0,Y 346.781,Z 654.735,A -85,B 0,C 180,E1 -14151.211,E2 -14151.211} C_VEL
LIN {X 0,Y 348.679,Z 643.374,A -85,B 0,C 180,E1 -14152.831,E2 -14152.831} C_VEL
LIN {X 0,Y 350.829,Z 629.856,A -85,B 0,C 180,E1 -14154.404,E2 -14154.404} C_VEL
LIN {X 0,Y 354.355,Z 606.866,A -85,B 0,C 180,E1 -14156.538,E2 -14156.538} C_VEL
LIN {X 0,Y 356.678,Z 592.224,A -85,B 0,C 180,E1 -14157.663,E2 -14157.663} C_VEL
LIN {X 0,Y 358.872,Z 576.674,A -85,B 0,C 180,E1 -14158.593,E2 -14158.593} C_VEL
LIN {X 0,Y 360.857,Z 559.833,A -85,B 0,C 180,E1 -14159.337,E2 -14159.337} C_VEL
LIN {X 0,Y 367.966,Z 480.08,A -85,B 0,C 180,E1 -14161.886,E2 -14161.886} C_VEL
LIN {X 0,Y 372.259,Z 438.327,A -85,B 0,C 180,E1 -14163.281,E2 -14163.281} C_VEL
LIN {X 0,Y 371.535,Z 427.223,A -85,B 0,C 180,E1 -14164.067,E2 -14164.067} C_VEL
LIN {X 0,Y 371.031,Z 425.174,A -85,B 0,C 180,E1 -14164.3,E2 -14164.3} C_VEL
LIN {X 0,Y 368.106,Z 419.069,A -85,B 0,C 180,E1 -14165.387,E2 -14165.387} C_VEL
LIN {X 0,Y 365.967,Z 415.068,A -85,B 0,C 180,E1 -14166.239,E2 -14166.239} C_VEL
LIN {X 0,Y 363.466,Z 410.602,A -85,B 0,C 180,E1 -14167.349,E2 -14167.349} C_VEL
LIN {X 0,Y 359.939,Z 405.059,A -85,B 0,C 180,E1 -14169.166,E2 -14169.166} C_VEL
LIN {X 0,Y 356.523,Z 400.207,A -85,B 0,C 180,E1 -14171.582,E2 -14171.582} C_VEL
LIN {X 0,Y 356.081,Z 399.426,A -85,B 0,C 180,E1 -14172.149,E2 -14172.149} C_VEL
LIN {X 0,Y 355.557,Z 397.917,A -85,B 0,C 180,E1 -14174.636,E2 -14174.636} C_VEL
LIN {X 0,Y 355.394,Z 397.77,A -85,B 0,C 180,E1 -14177.028,E2 -14177.028} C_VEL
LIN {X 0,Y 355.616,Z 398.657,A -85,B 0,C 180,E1 -14179.294,E2 -14179.294} C_VEL
LIN {X 0,Y 355.985,Z 399.87,A -85,B 0,C 180,E1 -14180.585,E2 -14180.585} C_VEL
LIN {X 0,Y 358.338,Z 403.676,A -85,B 0,C 180,E1 -14182.61,E2 -14182.61} C_VEL
LIN {X 0,Y 360.288,Z 406.572,A -85,B 0,C 180,E1 -14183.82,E2 -14183.82} C_VEL
LIN {X 0,Y 363.642,Z 412.32,A -85,B 0,C 180,E1 -14185.57,E2 -14185.57} C_VEL
LIN {X 0,Y 366.456,Z 417.76,A -85,B 0,C 180,E1 -14186.838,E2 -14186.838} C_VEL
LIN {X 0,Y 368.936,Z 423.05,A -85,B 0,C 180,E1 -14187.86,E2 -14187.86} C_VEL
LIN {X 0,Y 369.922,Z 425.503,A -85,B 0,C 180,E1 -14188.259,E2 -14188.259} C_VEL
LIN {X 0,Y 371.345,Z 436.38,A -85,B 0,C 180,E1 -14189.27,E2 -14189.27} C_VEL
LIN {X 0,Y 371.7,Z 441.969,A -85,B 0,C 180,E1 -14189.678,E2 -14189.678} C_VEL
LIN {X 0,Y 363.133,Z 520.661,A -85,B 0,C 180,E1 -14192.479,E2 -14192.479} C_VEL
LIN {X 0,Y 360.268,Z 550.223,A -85,B 0,C 180,E1 -14193.576,E2 -14193.576} C_VEL
LIN {X 0,Y 358.415,Z 565.429,A -85,B 0,C 180,E1 -14194.367,E2 -14194.367} C_VEL
LIN {X 0,Y 356.423,Z 580.044,A -85,B 0,C 180,E1 -14195.391,E2 -14195.391} C_VEL
LIN {X 0,Y 354.187,Z 594.101,A -85,B 0,C 180,E1 -14196.619,E2 -14196.619} C_VEL
LIN {X 0,Y 351.914,Z 607.01,A -85,B 0,C 180,E1 -14198.01,E2 -14198.01} C_VEL
LIN {X 0,Y 349.926,Z 617.764,A -85,B 0,C 180,E1 -14199.423,E2 -14199.423} C_VEL
LIN {X 0,Y 347.845,Z 628.604,A -85,B 0,C 180,E1 -14201.139,E2 -14201.139} C_VEL
LIN {X 0,Y 345.693,Z 638.766,A -85,B 0,C 180,E1 -14203.095,E2 -14203.095} C_VEL
LIN {X 0,Y 344.077,Z 646.476,A -85,B 0,C 180,E1 -14204.905,E2 -14204.905} C_VEL
LIN {X 0,Y 342.651,Z 653.59,A -85,B 0,C 180,E1 -14206.961,E2 -14206.961} C_VEL
LIN {X 0,Y 341.7,Z 658.565,A -85,B 0,C 180,E1 -14208.732,E2 -14208.732} C_VEL
LIN {X 0,Y 340.654,Z 663.681,A -85,B 0,C 180,E1 -14211.099,E2 -14211.099} C_VEL
LIN {X 0,Y 340.102,Z 666.518,A -85,B 0,C 180,E1 -14212.878,E2 -14212.878} C_VEL
LIN {X 0,Y 339.552,Z 668.963,A -85,B 0,C 180,E1 -14215.251,E2 -14215.251} C_VEL
LIN {X 0,Y 339.428,Z 669.943,A -85,B 0,C 180,E1 -14217.627,E2 -14217.627} C_VEL
LIN {X 0,Y 339.23,Z 669.496,A -85,B 0,C 180,E1 -14220,E2 -14220} C_VEL
LIN {X 0,Y 339.204,Z 667.598,A -85,B 0,C 180,E1 -14222.375,E2 -14222.375} C_VEL
LIN {X 0,Y 339.337,Z 664.208,A -85,B 0,C 180,E1 -14224.752,E2 -14224.752} C_VEL
LIN {X 0,Y 339.637,Z 659.244,A -85,B 0,C 180,E1 -14227.132,E2 -14227.132} C_VEL
LIN {X 0,Y 339.873,Z 654.343,A -85,B 0,C 180,E1 -14228.922,E2 -14228.922} C_VEL
LIN {X 0,Y 340.459,Z 647.282,A -85,B 0,C 180,E1 -14231.008,E2 -14231.008} C_VEL
LIN {X 0,Y 341.291,Z 638.52,A -85,B 0,C 180,E1 -14233.092,E2 -14233.092} C_VEL
LIN {X 0,Y 342.12,Z 629.093,A -85,B 0,C 180,E1 -14234.924,E2 -14234.924} C_VEL
LIN {X 0,Y 343.174,Z 618.277,A -85,B 0,C 180,E1 -14236.661,E2 -14236.661} C_VEL
LIN {X 0,Y 344.375,Z 605.996,A -85,B 0,C 180,E1 -14238.287,E2 -14238.287} C_VEL
LIN {X 0,Y 345.52,Z 593.839,A -85,B 0,C 180,E1 -14239.61,E2 -14239.61} C_VEL
LIN {X 0,Y 346.689,Z 580.685,A -85,B 0,C 180,E1 -14240.779,E2 -14240.779} C_VEL
LIN {X 0,Y 347.72,Z 566.075,A -85,B 0,C 180,E1 -14241.801,E2 -14241.801} C_VEL
LIN {X 0,Y 348.714,Z 550.119,A -85,B 0,C 180,E1 -14242.632,E2 -14242.632} C_VEL
LIN {X 0,Y 349.401,Z 535.195,A -85,B 0,C 180,E1 -14243.172,E2 -14243.172} C_VEL
LIN {X 0,Y 353.299,Z 433.06,A -85,B 0,C 180,E1 -14246.032,E2 -14246.032} C_VEL
LIN {X 0,Y 347.87,Z 397.999,A -85,B 0,C 180,E1 -14247.468,E2 -14247.468} C_VEL
LIN {X 0,Y 348.145,Z 395.31,A -85,B 0,C 180,E1 -14247.992,E2 -14247.992} C_VEL
LIN {X 0,Y 346.922,Z 389,A -85,B 0,C 180,E1 -14249.413,E2 -14249.413} C_VEL
LIN {X 0,Y 343.451,Z 373.867,A -85,B 0,C 180,E1 -14252.967,E2 -14252.967} C_VEL
LIN {X 0,Y 340.79,Z 362.853,A -85,B 0,C 180,E1 -14255.724,E2 -14255.724} C_VEL
LIN {X 0,Y 340.694,Z 362.673,A -85,B 0,C 180,E1 -14258.382,E2 -14258.382} C_VEL
LIN {X 0,Y 340.691,Z 362.651,A -85,B 0,C 180,E1 -14262.044,E2 -14262.044} C_VEL
LIN {X 0,Y 340.65,Z 362.663,A -85,B 0,C 180,E1 -14266.228,E2 -14266.228} C_VEL
LIN {X 0,Y 340.684,Z 362.835,A -85,B 0,C 180,E1 -14269.658,E2 -14269.658} C_VEL
LIN {X 0,Y 345.003,Z 375.677,A -85,B 0,C 180,E1 -14272.605,E2 -14272.605} C_VEL
LIN {X 0,Y 348.726,Z 388.427,A -85,B 0,C 180,E1 -14275.268,E2 -14275.268} C_VEL
LIN {X 0,Y 350.831,Z 396.424,A -85,B 0,C 180,E1 -14276.782,E2 -14276.782} C_VEL
LIN {X 0,Y 356.038,Z 408.235,A -85,B 0,C 180,E1 -14277.616,E2 -14277.616} C_VEL
LIN {X 0,Y 360.636,Z 432.82,A -85,B 0,C 180,E1 -14278.641,E2 -14278.641} C_VEL
LIN {X 0,Y 361.703,Z 439.137,A -85,B 0,C 180,E1 -14278.888,E2 -14278.888} C_VEL
LIN {X 0,Y 358.131,Z 562.912,A -85,B 0,C 180,E1 -14281.383,E2 -14281.383} C_VEL
LIN {X 0,Y 357.231,Z 578.226,A -85,B 0,C 180,E1 -14281.869,E2 -14281.869} C_VEL
LIN {X 0,Y 355.926,Z 593.084,A -85,B 0,C 180,E1 -14282.56,E2 -14282.56} C_VEL
LIN {X 0,Y 354.404,Z 606.936,A -85,B 0,C 180,E1 -14283.424,E2 -14283.424} C_VEL
LIN {X 0,Y 352.747,Z 620.174,A -85,B 0,C 180,E1 -14284.478,E2 -14284.478} C_VEL
LIN {X 0,Y 350.821,Z 633.143,A -85,B 0,C 180,E1 -14285.752,E2 -14285.752} C_VEL
LIN {X 0,Y 348.725,Z 646.162,A -85,B 0,C 180,E1 -14287.329,E2 -14287.329} C_VEL
LIN {X 0,Y 346.845,Z 657.049,A -85,B 0,C 180,E1 -14288.917,E2 -14288.917} C_VEL
LIN {X 0,Y 345.047,Z 667.114,A -85,B 0,C 180,E1 -14290.671,E2 -14290.671} C_VEL
LIN {X 0,Y 343.3,Z 676.93,A -85,B 0,C 180,E1 -14292.732,E2 -14292.732} C_VEL
LIN {X 0,Y 341.732,Z 685.932,A -85,B 0,C 180,E1 -14295.045,E2 -14295.045} C_VEL
LIN {X 0,Y 340.629,Z 693.544,A -85,B 0,C 180,E1 -14297.488,E2 -14297.488} C_VEL
LIN {X 0,Y 339.785,Z 699.433,A -85,B 0,C 180,E1 -14299.874,E2 -14299.874} C_VEL
LIN {X 0,Y 339.424,Z 702.913,A -85,B 0,C 180,E1 -14301.666,E2 -14301.666} C_VEL
LIN {X 0,Y 339.088,Z 706.628,A -85,B 0,C 180,E1 -14304.189,E2 -14304.189} C_VEL
LIN {X 0,Y 339.035,Z 708.806,A -85,B 0,C 180,E1 -14306.434,E2 -14306.434} C_VEL
LIN {X 0,Y 338.953,Z 709.996,A -85,B 0,C 180,E1 -14308.812,E2 -14308.812} C_VEL
LIN {X 0,Y 338.953,Z 710.009,A -85,B 0,C 180,E1 -14311.188,E2 -14311.188} C_VEL
LIN {X 0,Y 339.037,Z 708.871,A -85,B 0,C 180,E1 -14313.565,E2 -14313.565} C_VEL
LIN {X 0,Y 339.034,Z 708.025,A -85,B 0,C 180,E1 -14314.575,E2 -14314.575} C_VEL
LIN {X 0,Y 338.429,Z 707.099,A -85,B 0,C 180,E1 -14315.554,E2 -14315.554} C_VEL
LIN {X 0,Y 335.714,Z 705.151,A -85,B 0,C 180,E1 -14317.14,E2 -14317.14} C_VEL
LIN {X 0,Y 333.469,Z 703.217,A -85,B 0,C 180,E1 -14318.409,E2 -14318.409} C_VEL
LIN {X 0,Y 332.609,Z 701.568,A -85,B 0,C 180,E1 -14319.378,E2 -14319.378} C_VEL
LIN {X 0,Y 332.595,Z 700.918,A -85,B 0,C 180,E1 -14319.703,E2 -14319.703} C_VEL
LIN {X 0,Y 333.361,Z 695.396,A -85,B 0,C 180,E1 -14322.17,E2 -14322.17} C_VEL
LIN {X 0,Y 334.427,Z 688.434,A -85,B 0,C 180,E1 -14324.606,E2 -14324.606} C_VEL
LIN {X 0,Y 335.728,Z 680.981,A -85,B 0,C 180,E1 -14326.728,E2 -14326.728} C_VEL
LIN {X 0,Y 337.384,Z 672.004,A -85,B 0,C 180,E1 -14328.837,E2 -14328.837} C_VEL
LIN {X 0,Y 339.374,Z 661.718,A -85,B 0,C 180,E1 -14330.827,E2 -14330.827} C_VEL
LIN {X 0,Y 341.452,Z 650.005,A -85,B 0,C 180,E1 -14332.701,E2 -14332.701} C_VEL
LIN {X 0,Y 343.637,Z 637.77,A -85,B 0,C 180,E1 -14334.305,E2 -14334.305} C_VEL
LIN {X 0,Y 345.545,Z 625.781,A -85,B 0,C 180,E1 -14335.607,E2 -14335.607} C_VEL
LIN {X 0,Y 347.664,Z 611.031,A -85,B 0,C 180,E1 -14336.892,E2 -14336.892} C_VEL
LIN {X 0,Y 349.33,Z 596.467,A -85,B 0,C 180,E1 -14337.889,E2 -14337.889} C_VEL
LIN {X 0,Y 350.669,Z 582.948,A -85,B 0,C 180,E1 -14338.587,E2 -14338.587} C_VEL
LIN {X 0,Y 351.754,Z 567.764,A -85,B 0,C 180,E1 -14339.144,E2 -14339.144} C_VEL
LIN {X 0,Y 352.61,Z 541.839,A -85,B 0,C 180,E1 -14339.722,E2 -14339.722} C_VEL
LIN {X 0,Y 355.603,Z 439.488,A -85,B 0,C 180,E1 -14341.806,E2 -14341.806} C_VEL
LIN {X 0,Y 350.377,Z 410.981,A -85,B 0,C 180,E1 -14343.015,E2 -14343.015} C_VEL
LIN {X 0,Y 343.63,Z 396.013,A -85,B 0,C 180,E1 -14344.155,E2 -14344.155} C_VEL
LIN {X 0,Y 340,Z 382.873,A -85,B 0,C 180,E1 -14346.83,E2 -14346.83} C_VEL
LIN {X 0,Y 335.755,Z 369.968,A -85,B 0,C 180,E1 -14349.714,E2 -14349.714} C_VEL
LIN {X 0,Y 333.656,Z 363.704,A -85,B 0,C 180,E1 -14351.257,E2 -14351.257} C_VEL
LIN {X 0,Y 333.592,Z 363.555,A -85,B 0,C 180,E1 -14354.25,E2 -14354.25} C_VEL
LIN {X 0,Y 333.637,Z 363.546,A -85,B 0,C 180,E1 -14357.618,E2 -14357.618} C_VEL
LIN {X 0,Y 333.615,Z 363.546,A -85,B 0,C 180,E1 -14361.21,E2 -14361.21} C_VEL
LIN {X 0,Y 333.673,Z 363.538,A -85,B 0,C 180,E1 -14363.86,E2 -14363.86} C_VEL
LIN {X 0,Y 333.644,Z 363.543,A -85,B 0,C 180,E1 -14367.413,E2 -14367.413} C_VEL
LIN {X 0,Y 333.653,Z 363.549,A -85,B 0,C 180,E1 -14371.022,E2 -14371.022} C_VEL
LIN {X 0,Y 333.698,Z 363.543,A -85,B 0,C 180,E1 -14375.088,E2 -14375.088} C_VEL
LIN {X 0,Y 333.664,Z 363.538,A -85,B 0,C 180,E1 -14379.018,E2 -14379.018} C_VEL
LIN {X 0,Y 333.741,Z 363.53,A -85,B 0,C 180,E1 -14381.586,E2 -14381.586} C_VEL
LIN {X 0,Y 333.809,Z 363.529,A -85,B 0,C 180,E1 -14385.577,E2 -14385.577} C_VEL
LIN {X 0,Y 333.818,Z 363.506,A -85,B 0,C 180,E1 -14389.077,E2 -14389.077} C_VEL
LIN {X 0,Y 333.993,Z 363.505,A -85,B 0,C 180,E1 -14392.747,E2 -14392.747} C_VEL
LIN {X 0,Y 333.796,Z 363.508,A -85,B 0,C 180,E1 -14395.169,E2 -14395.169} C_VEL
LIN {X 0,Y 334.094,Z 363.492,A -85,B 0,C 180,E1 -14397.589,E2 -14397.589} C_VEL
LIN {X 0,Y 334.226,Z 363.466,A -85,B 0,C 180,E1 -14400,E2 -14400} C_VEL
LIN {X 0,Y 334.103,Z 363.475,A -85,B 0,C 180,E1 -14402.411,E2 -14402.411} C_VEL
LIN {X 0,Y 333.999,Z 363.497,A -85,B 0,C 180,E1 -14406.039,E2 -14406.039} C_VEL
LIN {X 0,Y 333.821,Z 363.52,A -85,B 0,C 180,E1 -14409.696,E2 -14409.696} C_VEL
LIN {X 0,Y 333.797,Z 363.508,A -85,B 0,C 180,E1 -14413.391,E2 -14413.391} C_VEL
LIN {X 0,Y 333.72,Z 363.541,A -85,B 0,C 180,E1 -14417.147,E2 -14417.147} C_VEL
LIN {X 0,Y 333.69,Z 363.524,A -85,B 0,C 180,E1 -14419.693,E2 -14419.693} C_VEL
LIN {X 0,Y 333.693,Z 363.543,A -85,B 0,C 180,E1 -14422.278,E2 -14422.278} C_VEL
LIN {X 0,Y 333.736,Z 363.532,A -85,B 0,C 180,E1 -14426.246,E2 -14426.246} C_VEL
LIN {X 0,Y 333.711,Z 363.531,A -85,B 0,C 180,E1 -14428.972,E2 -14428.972} C_VEL
LIN {X 0,Y 333.643,Z 363.552,A -85,B 0,C 180,E1 -14432.587,E2 -14432.587} C_VEL
LIN {X 0,Y 333.675,Z 363.546,A -85,B 0,C 180,E1 -14436.139,E2 -14436.139} C_VEL
LIN {X 0,Y 333.645,Z 363.507,A -85,B 0,C 180,E1 -14439.192,E2 -14439.192} C_VEL
LIN {X 0,Y 333.632,Z 363.534,A -85,B 0,C 180,E1 -14442.5,E2 -14442.5} C_VEL
LIN {X 0,Y 333.596,Z 363.522,A -85,B 0,C 180,E1 -14445.955,E2 -14445.955} C_VEL
LIN {X 0,Y 333.647,Z 363.55,A -85,B 0,C 180,E1 -14449.315,E2 -14449.315} C_VEL
LIN {X 0,Y 333.71,Z 363.733,A -85,B 0,C 180,E1 -14451.151,E2 -14451.151} C_VEL
LIN {X 0,Y 337.362,Z 377.385,A -85,B 0,C 180,E1 -14454.237,E2 -14454.237} C_VEL
LIN {X 0,Y 342.775,Z 392.175,A -85,B 0,C 180,E1 -14456.01,E2 -14456.01} C_VEL
LIN {X 0,Y 350.605,Z 409.495,A -85,B 0,C 180,E1 -14457.287,E2 -14457.287} C_VEL
LIN {X 0,Y 351.58,Z 414.028,A -85,B 0,C 180,E1 -14457.497,E2 -14457.497} C_VEL
LIN {X 0,Y 355.041,Z 437.475,A -85,B 0,C 180,E1 -14458.401,E2 -14458.401} C_VEL
LIN {X 0,Y 351.338,Z 563.616,A -85,B 0,C 180,E1 -14460.982,E2 -14460.982} C_VEL
LIN {X 0,Y 350.394,Z 578.541,A -85,B 0,C 180,E1 -14461.47,E2 -14461.47} C_VEL
LIN {X 0,Y 349.111,Z 593.174,A -85,B 0,C 180,E1 -14462.174,E2 -14462.174} C_VEL
LIN {X 0,Y 347.643,Z 606.674,A -85,B 0,C 180,E1 -14463.043,E2 -14463.043} C_VEL
LIN {X 0,Y 345.682,Z 621.281,A -85,B 0,C 180,E1 -14464.242,E2 -14464.242} C_VEL
LIN {X 0,Y 343.681,Z 633.943,A -85,B 0,C 180,E1 -14465.538,E2 -14465.538} C_VEL
LIN {X 0,Y 341.538,Z 646.709,A -85,B 0,C 180,E1 -14467.145,E2 -14467.145} C_VEL
LIN {X 0,Y 339.72,Z 657.174,A -85,B 0,C 180,E1 -14468.739,E2 -14468.739} C_VEL
LIN {X 0,Y 337.845,Z 667.226,A -85,B 0,C 180,E1 -14470.559,E2 -14470.559} C_VEL
LIN {X 0,Y 336.079,Z 676.845,A -85,B 0,C 180,E1 -14472.663,E2 -14472.663} C_VEL
LIN {X 0,Y 334.655,Z 685.044,A -85,B 0,C 180,E1 -14474.844,E2 -14474.844} C_VEL
LIN {X 0,Y 333.551,Z 692.292,A -85,B 0,C 180,E1 -14477.218,E2 -14477.218} C_VEL
LIN {X 0,Y 332.707,Z 698.196,A -85,B 0,C 180,E1 -14479.657,E2 -14479.657} C_VEL
LIN {X 0,Y 332.351,Z 701.679,A -85,B 0,C 180,E1 -14481.488,E2 -14481.488} C_VEL
LIN {X 0,Y 332.02,Z 705.529,A -85,B 0,C 180,E1 -14484.191,E2 -14484.191} C_VEL
LIN {X 0,Y 331.955,Z 707.538,A -85,B 0,C 180,E1 -14486.359,E2 -14486.359} C_VEL
LIN {X 0,Y 331.874,Z 708.707,A -85,B 0,C 180,E1 -14488.787,E2 -14488.787} C_VEL
LIN {X 0,Y 331.875,Z 708.706,A -85,B 0,C 180,E1 -14491.214,E2 -14491.214} C_VEL
LIN {X 0,Y 331.956,Z 707.533,A -85,B 0,C 180,E1 -14493.642,E2 -14493.642} C_VEL
LIN {X 0,Y 332.042,Z 705.2,A -85,B 0,C 180,E1 -14496.075,E2 -14496.075} C_VEL
LIN {X 0,Y 332.351,Z 701.652,A -85,B 0,C 180,E1 -14498.513,E2 -14498.513} C_VEL
LIN {X 0,Y 332.85,Z 696.805,A -85,B 0,C 180,E1 -14500.955,E2 -14500.955} C_VEL
LIN {X 0,Y 333.8,Z 690.533,A -85,B 0,C 180,E1 -14503.391,E2 -14503.391} C_VEL
LIN {X 0,Y 335.058,Z 682.642,A -85,B 0,C 180,E1 -14505.824,E2 -14505.824} C_VEL
LIN {X 0,Y 336.558,Z 674.208,A -85,B 0,C 180,E1 -14507.94,E2 -14507.94} C_VEL
LIN {X 0,Y 338.154,Z 665.652,A -85,B 0,C 180,E1 -14509.739,E2 -14509.739} C_VEL
LIN {X 0,Y 340.009,Z 655.407,A -85,B 0,C 180,E1 -14511.542,E2 -14511.542} C_VEL
LIN {X 0,Y 342.128,Z 643.394,A -85,B 0,C 180,E1 -14513.293,E2 -14513.293} C_VEL
LIN {X 0,Y 344.164,Z 631.241,A -85,B 0,C 180,E1 -14514.748,E2 -14514.748} C_VEL
LIN {X 0,Y 347.847,Z 610.888,A -85,B 0,C 180,E1 -14516.864,E2 -14516.864} C_VEL
LIN {X 0,Y 350.284,Z 597.188,A -85,B 0,C 180,E1 -14518.018,E2 -14518.018} C_VEL
LIN {X 0,Y 352.723,Z 581.707,A -85,B 0,C 180,E1 -14519.057,E2 -14519.057} C_VEL
LIN {X 0,Y 354.953,Z 565.51,A -85,B 0,C 180,E1 -14519.874,E2 -14519.874} C_VEL
LIN {X 0,Y 356.903,Z 546.526,A -85,B 0,C 180,E1 -14520.55,E2 -14520.55} C_VEL
LIN {X 0,Y 363.295,Z 480.686,A -85,B 0,C 180,E1 -14522.715,E2 -14522.715} C_VEL
LIN {X 0,Y 367.854,Z 439.519,A -85,B 0,C 180,E1 -14524.138,E2 -14524.138} C_VEL
LIN {X 0,Y 367.312,Z 430.07,A -85,B 0,C 180,E1 -14524.853,E2 -14524.853} C_VEL
LIN {X 0,Y 364.615,Z 424.173,A -85,B 0,C 180,E1 -14525.948,E2 -14525.948} C_VEL
LIN {X 0,Y 362.229,Z 419.559,A -85,B 0,C 180,E1 -14526.995,E2 -14526.995} C_VEL
LIN {X 0,Y 360.357,Z 416.135,A -85,B 0,C 180,E1 -14527.905,E2 -14527.905} C_VEL
LIN {X 0,Y 357.498,Z 411.328,A -85,B 0,C 180,E1 -14529.525,E2 -14529.525} C_VEL
LIN {X 0,Y 354.262,Z 406.529,A -85,B 0,C 180,E1 -14532.02,E2 -14532.02} C_VEL
LIN {X 0,Y 352.589,Z 404.537,A -85,B 0,C 180,E1 -14534.146,E2 -14534.146} C_VEL
LIN {X 0,Y 352.043,Z 403.911,A -85,B 0,C 180,E1 -14535.946,E2 -14535.946} C_VEL
LIN {X 0,Y 352.316,Z 404.394,A -85,B 0,C 180,E1 -14537.994,E2 -14537.994} C_VEL
LIN {X 0,Y 353.678,Z 406.155,A -85,B 0,C 180,E1 -14540.126,E2 -14540.126} C_VEL
LIN {X 0,Y 356.116,Z 410.227,A -85,B 0,C 180,E1 -14542.364,E2 -14542.364} C_VEL
LIN {X 0,Y 357.826,Z 412.952,A -85,B 0,C 180,E1 -14543.507,E2 -14543.507} C_VEL
LIN {X 0,Y 360.899,Z 418.612,A -85,B 0,C 180,E1 -14545.243,E2 -14545.243} C_VEL
LIN {X 0,Y 363.418,Z 423.744,A -85,B 0,C 180,E1 -14546.46,E2 -14546.46} C_VEL
LIN {X 0,Y 366,Z 429.648,A -85,B 0,C 180,E1 -14547.599,E2 -14547.599} C_VEL
LIN {X 0,Y 367.065,Z 439.687,A -85,B 0,C 180,E1 -14548.548,E2 -14548.548} C_VEL
LIN {X 0,Y 367.286,Z 443.37,A -85,B 0,C 180,E1 -14548.839,E2 -14548.839} C_VEL
LIN {X 0,Y 357.774,Z 524.28,A -85,B 0,C 180,E1 -14551.792,E2 -14551.792} C_VEL
LIN {X 0,Y 354.863,Z 551.909,A -85,B 0,C 180,E1 -14552.862,E2 -14552.862} C_VEL
LIN {X 0,Y 352.799,Z 567.699,A -85,B 0,C 180,E1 -14553.746,E2 -14553.746} C_VEL
LIN {X 0,Y 350.627,Z 582.158,A -85,B 0,C 180,E1 -14554.805,E2 -14554.805} C_VEL
LIN {X 0,Y 348.266,Z 595.739,A -85,B 0,C 180,E1 -14556.039,E2 -14556.039} C_VEL
LIN {X 0,Y 345.845,Z 608.341,A -85,B 0,C 180,E1 -14557.446,E2 -14557.446} C_VEL
LIN {X 0,Y 343.534,Z 619.826,A -85,B 0,C 180,E1 -14559.022,E2 -14559.022} C_VEL
LIN {X 0,Y 341.352,Z 630.321,A -85,B 0,C 180,E1 -14560.767,E2 -14560.767} C_VEL
LIN {X 0,Y 339.191,Z 639.685,A -85,B 0,C 180,E1 -14562.632,E2 -14562.632} C_VEL
LIN {X 0,Y 337.347,Z 647.743,A -85,B 0,C 180,E1 -14564.596,E2 -14564.596} C_VEL
LIN {X 0,Y 335.821,Z 654.682,A -85,B 0,C 180,E1 -14566.691,E2 -14566.691} C_VEL
LIN {X 0,Y 334.797,Z 659.498,A -85,B 0,C 180,E1 -14568.497,E2 -14568.497} C_VEL
LIN {X 0,Y 333.698,Z 664.465,A -85,B 0,C 180,E1 -14570.912,E2 -14570.912} C_VEL
LIN {X 0,Y 333.086,Z 667.19,A -85,B 0,C 180,E1 -14572.727,E2 -14572.727} C_VEL
LIN {X 0,Y 332.494,Z 669.493,A -85,B 0,C 180,E1 -14575.15,E2 -14575.15} C_VEL
LIN {X 0,Y 332.342,Z 670.351,A -85,B 0,C 180,E1 -14577.576,E2 -14577.576} C_VEL
LIN {X 0,Y 332.137,Z 669.781,A -85,B 0,C 180,E1 -14580,E2 -14580} C_VEL
LIN {X 0,Y 332.112,Z 667.761,A -85,B 0,C 180,E1 -14582.426,E2 -14582.426} C_VEL
LIN {X 0,Y 332.258,Z 664.244,A -85,B 0,C 180,E1 -14584.854,E2 -14584.854} C_VEL
LIN {X 0,Y 332.522,Z 659.718,A -85,B 0,C 180,E1 -14587.026,E2 -14587.026} C_VEL
LIN {X 0,Y 332.821,Z 654.106,A -85,B 0,C 180,E1 -14589.113,E2 -14589.113} C_VEL
LIN {X 0,Y 333.415,Z 646.883,A -85,B 0,C 180,E1 -14591.244,E2 -14591.244} C_VEL
LIN {X 0,Y 334.301,Z 637.884,A -85,B 0,C 180,E1 -14593.371,E2 -14593.371} C_VEL
LIN {X 0,Y 335.199,Z 627.816,A -85,B 0,C 180,E1 -14595.319,E2 -14595.319} C_VEL
LIN {X 0,Y 336.398,Z 616.201,A -85,B 0,C 180,E1 -14597.164,E2 -14597.164} C_VEL
LIN {X 0,Y 337.484,Z 604.682,A -85,B 0,C 180,E1 -14598.674,E2 -14598.674} C_VEL
LIN {X 0,Y 338.764,Z 592.199,A -85,B 0,C 180,E1 -14600.018,E2 -14600.018} C_VEL
LIN {X 0,Y 339.907,Z 579.279,A -85,B 0,C 180,E1 -14601.15,E2 -14601.15} C_VEL
LIN {X 0,Y 340.95,Z 564.465,A -85,B 0,C 180,E1 -14602.178,E2 -14602.178} C_VEL
LIN {X 0,Y 341.893,Z 549.612,A -85,B 0,C 180,E1 -14602.95,E2 -14602.95} C_VEL
LIN {X 0,Y 342.6,Z 534.445,A -85,B 0,C 180,E1 -14603.499,E2 -14603.499} C_VEL
LIN {X 0,Y 346.652,Z 434.598,A -85,B 0,C 180,E1 -14606.377,E2 -14606.377} C_VEL
LIN {X 0,Y 341.13,Z 398.177,A -85,B 0,C 180,E1 -14607.902,E2 -14607.902} C_VEL
LIN {X 0,Y 341.219,Z 396.134,A -85,B 0,C 180,E1 -14608.277,E2 -14608.277} C_VEL
LIN {X 0,Y 338.359,Z 383.276,A -85,B 0,C 180,E1 -14611.283,E2 -14611.283} C_VEL
LIN {X 0,Y 335.308,Z 370.266,A -85,B 0,C 180,E1 -14614.466,E2 -14614.466} C_VEL
LIN {X 0,Y 333.723,Z 363.825,A -85,B 0,C 180,E1 -14616.133,E2 -14616.133} C_VEL
LIN {X 0,Y 333.662,Z 363.549,A -85,B 0,C 180,E1 -14616.831,E2 -14616.831} C_VEL
LIN {X 0,Y 333.603,Z 363.553,A -85,B 0,C 180,E1 -14620.774,E2 -14620.774} C_VEL
LIN {X 0,Y 333.591,Z 363.549,A -85,B 0,C 180,E1 -14624.25,E2 -14624.25} C_VEL
LIN {X 0,Y 333.638,Z 363.546,A -85,B 0,C 180,E1 -14628.43,E2 -14628.43} C_VEL
LIN {X 0,Y 333.674,Z 363.829,A -85,B 0,C 180,E1 -14628.923,E2 -14628.923} C_VEL
LIN {X 0,Y 338.331,Z 377.522,A -85,B 0,C 180,E1 -14632.126,E2 -14632.126} C_VEL
LIN {X 0,Y 342.156,Z 390.53,A -85,B 0,C 180,E1 -14634.891,E2 -14634.891} C_VEL
LIN {X 0,Y 343.774,Z 396.501,A -85,B 0,C 180,E1 -14636.018,E2 -14636.018} C_VEL
LIN {X 0,Y 350.41,Z 411.364,A -85,B 0,C 180,E1 -14637.108,E2 -14637.108} C_VEL
LIN {X 0,Y 355.16,Z 437.337,A -85,B 0,C 180,E1 -14638.209,E2 -14638.209} C_VEL
LIN {X 0,Y 355.606,Z 440.377,A -85,B 0,C 180,E1 -14638.324,E2 -14638.324} C_VEL
LIN {X 0,Y 351.875,Z 564.199,A -85,B 0,C 180,E1 -14640.867,E2 -14640.867} C_VEL
LIN {X 0,Y 350.908,Z 579.125,A -85,B 0,C 180,E1 -14641.36,E2 -14641.36} C_VEL
LIN {X 0,Y 349.514,Z 594.171,A -85,B 0,C 180,E1 -14642.087,E2 -14642.087} C_VEL
LIN {X 0,Y 347.849,Z 609.023,A -85,B 0,C 180,E1 -14643.061,E2 -14643.061} C_VEL
LIN {X 0,Y 345.885,Z 623.234,A -85,B 0,C 180,E1 -14644.258,E2 -14644.258} C_VEL
LIN {X 0,Y 343.904,Z 635.649,A -85,B 0,C 180,E1 -14645.554,E2 -14645.554} C_VEL
LIN {X 0,Y 341.748,Z 648.244,A -85,B 0,C 180,E1 -14647.16,E2 -14647.16} C_VEL
LIN {X 0,Y 339.902,Z 658.66,A -85,B 0,C 180,E1 -14648.76,E2 -14648.76} C_VEL
LIN {X 0,Y 337.991,Z 668.58,A -85,B 0,C 180,E1 -14650.567,E2 -14650.567} C_VEL
LIN {X 0,Y 336.243,Z 678.142,A -85,B 0,C 180,E1 -14652.671,E2 -14652.671} C_VEL
LIN {X 0,Y 334.81,Z 685.989,A -85,B 0,C 180,E1 -14654.75,E2 -14654.75} C_VEL
LIN {X 0,Y 333.643,Z 693.53,A -85,B 0,C 180,E1 -14657.222,E2 -14657.222} C_VEL
LIN {X 0,Y 332.748,Z 699.42,A -85,B 0,C 180,E1 -14659.657,E2 -14659.657} C_VEL
LIN {X 0,Y 332.356,Z 702.9,A -85,B 0,C 180,E1 -14661.488,E2 -14661.488} C_VEL
LIN {X 0,Y 332.013,Z 706.782,A -85,B 0,C 180,E1 -14664.205,E2 -14664.205} C_VEL
LIN {X 0,Y 331.939,Z 708.793,A -85,B 0,C 180,E1 -14666.358,E2 -14666.358} C_VEL
LIN {X 0,Y 331.862,Z 709.982,A -85,B 0,C 180,E1 -14668.786,E2 -14668.786} C_VEL
LIN {X 0,Y 331.862,Z 709.995,A -85,B 0,C 180,E1 -14671.213,E2 -14671.213} C_VEL
LIN {X 0,Y 331.942,Z 708.857,A -85,B 0,C 180,E1 -14673.642,E2 -14673.642} C_VEL
LIN {X 0,Y 332.043,Z 706.569,A -85,B 0,C 180,E1 -14676.075,E2 -14676.075} C_VEL
LIN {X 0,Y 332.358,Z 703.082,A -85,B 0,C 180,E1 -14678.512,E2 -14678.512} C_VEL
LIN {X 0,Y 332.595,Z 700.918,A -85,B 0,C 180,E1 -14679.703,E2 -14679.703} C_VEL
LIN {X 0,Y 332.171,Z 699.015,A -85,B 0,C 180,E1 -14680.665,E2 -14680.665} C_VEL
LIN {X 0,Y 329.821,Z 695.618,A -85,B 0,C 180,E1 -14682.227,E2 -14682.227} C_VEL
LIN {X 0,Y 327.594,Z 691.754,A -85,B 0,C 180,E1 -14683.776,E2 -14683.776} C_VEL
LIN {X 0,Y 327.372,Z 689.088,A -85,B 0,C 180,E1 -14684.702,E2 -14684.702} C_VEL
LIN {X 0,Y 328.638,Z 682.107,A -85,B 0,C 180,E1 -14686.78,E2 -14686.78} C_VEL
LIN {X 0,Y 330.341,Z 673.344,A -85,B 0,C 180,E1 -14688.932,E2 -14688.932} C_VEL
LIN {X 0,Y 332.172,Z 664.411,A -85,B 0,C 180,E1 -14690.756,E2 -14690.756} C_VEL
LIN {X 0,Y 334.127,Z 653.884,A -85,B 0,C 180,E1 -14692.573,E2 -14692.573} C_VEL
LIN {X 0,Y 336.309,Z 642.421,A -85,B 0,C 180,E1 -14694.212,E2 -14694.212} C_VEL
LIN {X 0,Y 338.446,Z 629.938,A -85,B 0,C 180,E1 -14695.688,E2 -14695.688} C_VEL
LIN {X 0,Y 340.575,Z 616.245,A -85,B 0,C 180,E1 -14697,E2 -14697} C_VEL
LIN {X 0,Y 342.391,Z 602.644,A -85,B 0,C 180,E1 -14698.039,E2 -14698.039} C_VEL
LIN {X 0,Y 343.874,Z 587.983,A -85,B 0,C 180,E1 -14698.913,E2 -14698.913} C_VEL
LIN {X 0,Y 345.196,Z 572.999,A -85,B 0,C 180,E1 -14699.543,E2 -14699.543} C_VEL
LIN {X 0,Y 346.018,Z 557.692,A -85,B 0,C 180,E1 -14699.968,E2 -14699.968} C_VEL
LIN {X 0,Y 349.555,Z 440.774,A -85,B 0,C 180,E1 -14702.388,E2 -14702.388} C_VEL
LIN {X 0,Y 344.66,Z 413.849,A -85,B 0,C 180,E1 -14703.561,E2 -14703.561} C_VEL
LIN {X 0,Y 337.319,Z 397.751,A -85,B 0,C 180,E1 -14704.795,E2 -14704.795} C_VEL
LIN {X 0,Y 336.474,Z 395.66,A -85,B 0,C 180,E1 -14705.022,E2 -14705.022} C_VEL
LIN {X 0,Y 332.456,Z 381.8,A -85,B 0,C 180,E1 -14707.968,E2 -14707.968} C_VEL
LIN {X 0,Y 328.3,Z 369.505,A -85,B 0,C 180,E1 -14710.829,E2 -14710.829} C_VEL
LIN {X 0,Y 326.628,Z 364.641,A -85,B 0,C 180,E1 -14712.062,E2 -14712.062} C_VEL
LIN {X 0,Y 326.526,Z 364.432,A -85,B 0,C 180,E1 -14715.257,E2 -14715.257} C_VEL
LIN {X 0,Y 326.562,Z 364.428,A -85,B 0,C 180,E1 -14718.152,E2 -14718.152} C_VEL
LIN {X 0,Y 326.566,Z 364.424,A -85,B 0,C 180,E1 -14721.383,E2 -14721.383} C_VEL
LIN {X 0,Y 326.617,Z 364.414,A -85,B 0,C 180,E1 -14724.852,E2 -14724.852} C_VEL
LIN {X 0,Y 326.608,Z 364.418,A -85,B 0,C 180,E1 -14727.455,E2 -14727.455} C_VEL
LIN {X 0,Y 326.616,Z 364.426,A -85,B 0,C 180,E1 -14730.336,E2 -14730.336} C_VEL
LIN {X 0,Y 326.642,Z 364.42,A -85,B 0,C 180,E1 -14734.644,E2 -14734.644} C_VEL
LIN {X 0,Y 326.614,Z 364.411,A -85,B 0,C 180,E1 -14738.543,E2 -14738.543} C_VEL
LIN {X 0,Y 326.707,Z 364.412,A -85,B 0,C 180,E1 -14741.175,E2 -14741.175} C_VEL
LIN {X 0,Y 326.763,Z 364.404,A -85,B 0,C 180,E1 -14745.433,E2 -14745.433} C_VEL
LIN {X 0,Y 326.758,Z 364.385,A -85,B 0,C 180,E1 -14748.838,E2 -14748.838} C_VEL
LIN {X 0,Y 326.943,Z 364.383,A -85,B 0,C 180,E1 -14752.589,E2 -14752.589} C_VEL
LIN {X 0,Y 326.982,Z 364.366,A -85,B 0,C 180,E1 -14753.831,E2 -14753.831} C_VEL
LIN {X 0,Y 327.034,Z 364.37,A -85,B 0,C 180,E1 -14757.537,E2 -14757.537} C_VEL
LIN {X 0,Y 327.178,Z 364.344,A -85,B 0,C 180,E1 -14760,E2 -14760} C_VEL
LIN {X 0,Y 327.043,Z 364.354,A -85,B 0,C 180,E1 -14762.463,E2 -14762.463} C_VEL
LIN {X 0,Y 326.953,Z 364.374,A -85,B 0,C 180,E1 -14766.17,E2 -14766.17} C_VEL
LIN {X 0,Y 326.784,Z 364.4,A -85,B 0,C 180,E1 -14769.907,E2 -14769.907} C_VEL
LIN {X 0,Y 326.759,Z 364.383,A -85,B 0,C 180,E1 -14773.685,E2 -14773.685} C_VEL
LIN {X 0,Y 326.664,Z 364.415,A -85,B 0,C 180,E1 -14777.53,E2 -14777.53} C_VEL
LIN {X 0,Y 326.636,Z 364.404,A -85,B 0,C 180,E1 -14780.137,E2 -14780.137} C_VEL
LIN {X 0,Y 326.621,Z 364.426,A -85,B 0,C 180,E1 -14782.787,E2 -14782.787} C_VEL
LIN {X 0,Y 326.69,Z 364.4,A -85,B 0,C 180,E1 -14785.484,E2 -14785.484} C_VEL
LIN {X 0,Y 326.66,Z 364.404,A -85,B 0,C 180,E1 -14789.659,E2 -14789.659} C_VEL
LIN {X 0,Y 326.606,Z 364.414,A -85,B 0,C 180,E1 -14794.019,E2 -14794.019} C_VEL
LIN {X 0,Y 326.627,Z 364.419,A -85,B 0,C 180,E1 -14797.238,E2 -14797.238} C_VEL
LIN {X 0,Y 326.576,Z 364.384,A -85,B 0,C 180,E1 -14801.131,E2 -14801.131} C_VEL
LIN {X 0,Y 326.527,Z 364.422,A -85,B 0,C 180,E1 -14804.743,E2 -14804.743} C_VEL
LIN {X 0,Y 326.575,Z 364.403,A -85,B 0,C 180,E1 -14808.154,E2 -14808.154} C_VEL
LIN {X 0,Y 326.655,Z 364.664,A -85,B 0,C 180,E1 -14810.673,E2 -14810.673} C_VEL
LIN {X 0,Y 329.147,Z 373.91,A -85,B 0,C 180,E1 -14812.856,E2 -14812.856} C_VEL
LIN {X 0,Y 335.796,Z 392.028,A -85,B 0,C 180,E1 -14815.195,E2 -14815.195} C_VEL
LIN {X 0,Y 345.18,Z 412.885,A -85,B 0,C 180,E1 -14816.786,E2 -14816.786} C_VEL
LIN {X 0,Y 349.001,Z 438.157,A -85,B 0,C 180,E1 -14817.801,E2 -14817.801} C_VEL
LIN {X 0,Y 345.157,Z 563.734,A -85,B 0,C 180,E1 -14820.411,E2 -14820.411} C_VEL
LIN {X 0,Y 344.191,Z 578.614,A -85,B 0,C 180,E1 -14820.907,E2 -14820.907} C_VEL
LIN {X 0,Y 342.844,Z 593.227,A -85,B 0,C 180,E1 -14821.62,E2 -14821.62} C_VEL
LIN {X 0,Y 341.241,Z 607.277,A -85,B 0,C 180,E1 -14822.542,E2 -14822.542} C_VEL
LIN {X 0,Y 339.295,Z 621.315,A -85,B 0,C 180,E1 -14823.721,E2 -14823.721} C_VEL
LIN {X 0,Y 337.206,Z 633.973,A -85,B 0,C 180,E1 -14825.036,E2 -14825.036} C_VEL
LIN {X 0,Y 334.967,Z 646.735,A -85,B 0,C 180,E1 -14826.671,E2 -14826.671} C_VEL
LIN {X 0,Y 332.945,Z 657.839,A -85,B 0,C 180,E1 -14828.403,E2 -14828.403} C_VEL
LIN {X 0,Y 331.125,Z 667.247,A -85,B 0,C 180,E1 -14830.148,E2 -14830.148} C_VEL
LIN {X 0,Y 329.236,Z 676.864,A -85,B 0,C 180,E1 -14832.291,E2 -14832.291} C_VEL
LIN {X 0,Y 327.788,Z 684.864,A -85,B 0,C 180,E1 -14834.455,E2 -14834.455} C_VEL
LIN {X 0,Y 326.573,Z 692.308,A -85,B 0,C 180,E1 -14836.941,E2 -14836.941} C_VEL
LIN {X 0,Y 325.681,Z 698.212,A -85,B 0,C 180,E1 -14839.431,E2 -14839.431} C_VEL
LIN {X 0,Y 325.302,Z 701.695,A -85,B 0,C 180,E1 -14841.302,E2 -14841.302} C_VEL
LIN {X 0,Y 324.957,Z 705.228,A -85,B 0,C 180,E1 -14843.792,E2 -14843.792} C_VEL
LIN {X 0,Y 324.862,Z 707.553,A -85,B 0,C 180,E1 -14846.279,E2 -14846.279} C_VEL
LIN {X 0,Y 324.786,Z 708.721,A -85,B 0,C 180,E1 -14848.76,E2 -14848.76} C_VEL
LIN {X 0,Y 324.787,Z 708.72,A -85,B 0,C 180,E1 -14851.24,E2 -14851.24} C_VEL
LIN {X 0,Y 324.863,Z 707.547,A -85,B 0,C 180,E1 -14853.721,E2 -14853.721} C_VEL
LIN {X 0,Y 324.957,Z 705.214,A -85,B 0,C 180,E1 -14856.208,E2 -14856.208} C_VEL
LIN {X 0,Y 325.302,Z 701.666,A -85,B 0,C 180,E1 -14858.698,E2 -14858.698} C_VEL
LIN {X 0,Y 325.831,Z 696.819,A -85,B 0,C 180,E1 -14861.194,E2 -14861.194} C_VEL
LIN {X 0,Y 326.823,Z 690.547,A -85,B 0,C 180,E1 -14863.683,E2 -14863.683} C_VEL
LIN {X 0,Y 328.174,Z 682.657,A -85,B 0,C 180,E1 -14866.165,E2 -14866.165} C_VEL
LIN {X 0,Y 329.754,Z 674.224,A -85,B 0,C 180,E1 -14868.323,E2 -14868.323} C_VEL
LIN {X 0,Y 331.45,Z 665.669,A -85,B 0,C 180,E1 -14870.155,E2 -14870.155} C_VEL
LIN {X 0,Y 333.496,Z 654.886,A -85,B 0,C 180,E1 -14872.08,E2 -14872.08} C_VEL
LIN {X 0,Y 335.602,Z 643.414,A -85,B 0,C 180,E1 -14873.774,E2 -14873.774} C_VEL
LIN {X 0,Y 339.802,Z 622.33,A -85,B 0,C 180,E1 -14876.403,E2 -14876.403} C_VEL
LIN {X 0,Y 342.845,Z 607.391,A -85,B 0,C 180,E1 -14877.923,E2 -14877.923} C_VEL
LIN {X 0,Y 345.438,Z 593.434,A -85,B 0,C 180,E1 -14879.061,E2 -14879.061} C_VEL
LIN {X 0,Y 347.851,Z 578.914,A -85,B 0,C 180,E1 -14880.004,E2 -14880.004} C_VEL
LIN {X 0,Y 350.329,Z 561.259,A -85,B 0,C 180,E1 -14880.852,E2 -14880.852} C_VEL
LIN {X 0,Y 359.632,Z 474.585,A -85,B 0,C 180,E1 -14883.819,E2 -14883.819} C_VEL
LIN {X 0,Y 363.682,Z 441.292,A -85,B 0,C 180,E1 -14884.999,E2 -14884.999} C_VEL
LIN {X 0,Y 363.362,Z 434.163,A -85,B 0,C 180,E1 -14885.565,E2 -14885.565} C_VEL
LIN {X 0,Y 360.4,Z 427.413,A -85,B 0,C 180,E1 -14886.916,E2 -14886.916} C_VEL
LIN {X 0,Y 357.704,Z 422.296,A -85,B 0,C 180,E1 -14888.285,E2 -14888.285} C_VEL
LIN {X 0,Y 355.02,Z 417.526,A -85,B 0,C 180,E1 -14889.93,E2 -14889.93} C_VEL
LIN {X 0,Y 352.099,Z 412.974,A -85,B 0,C 180,E1 -14892.394,E2 -14892.394} C_VEL
LIN {X 0,Y 350.643,Z 411.193,A -85,B 0,C 180,E1 -14894.549,E2 -14894.549} C_VEL
LIN {X 0,Y 350.231,Z 410.804,A -85,B 0,C 180,E1 -14896.254,E2 -14896.254} C_VEL
LIN {X 0,Y 350.655,Z 411.488,A -85,B 0,C 180,E1 -14898.296,E2 -14898.296} C_VEL
LIN {X 0,Y 351.794,Z 413.029,A -85,B 0,C 180,E1 -14900.055,E2 -14900.055} C_VEL
LIN {X 0,Y 354.582,Z 417.833,A -85,B 0,C 180,E1 -14902.622,E2 -14902.622} C_VEL
LIN {X 0,Y 357.714,Z 423.754,A -85,B 0,C 180,E1 -14904.624,E2 -14904.624} C_VEL
LIN {X 0,Y 360.332,Z 429.591,A -85,B 0,C 180,E1 -14906.035,E2 -14906.035} C_VEL
LIN {X 0,Y 362.25,Z 434.335,A -85,B 0,C 180,E1 -14906.969,E2 -14906.969} C_VEL
LIN {X 0,Y 363.072,Z 444.89,A -85,B 0,C 180,E1 -14907.965,E2 -14907.965} C_VEL
LIN {X 0,Y 352.539,Z 528.34,A -85,B 0,C 180,E1 -14911.09,E2 -14911.09} C_VEL
LIN {X 0,Y 349.763,Z 552.586,A -85,B 0,C 180,E1 -14912.068,E2 -14912.068} C_VEL
LIN {X 0,Y 347.572,Z 567.922,A -85,B 0,C 180,E1 -14912.938,E2 -14912.938} C_VEL
LIN {X 0,Y 345.063,Z 583.525,A -85,B 0,C 180,E1 -14914.118,E2 -14914.118} C_VEL
LIN {X 0,Y 342.409,Z 597.562,A -85,B 0,C 180,E1 -14915.441,E2 -14915.441} C_VEL
LIN {X 0,Y 339.601,Z 610.878,A -85,B 0,C 180,E1 -14917.007,E2 -14917.007} C_VEL
LIN {X 0,Y 337.174,Z 621.97,A -85,B 0,C 180,E1 -14918.607,E2 -14918.607} C_VEL
LIN {X 0,Y 334.877,Z 632.145,A -85,B 0,C 180,E1 -14920.38,E2 -14920.38} C_VEL
LIN {X 0,Y 332.734,Z 640.697,A -85,B 0,C 180,E1 -14922.153,E2 -14922.153} C_VEL
LIN {X 0,Y 330.636,Z 649.082,A -85,B 0,C 180,E1 -14924.276,E2 -14924.276} C_VEL
LIN {X 0,Y 329.005,Z 655.829,A -85,B 0,C 180,E1 -14926.41,E2 -14926.41} C_VEL
LIN {X 0,Y 327.903,Z 660.477,A -85,B 0,C 180,E1 -14928.252,E2 -14928.252} C_VEL
LIN {X 0,Y 326.75,Z 665.28,A -85,B 0,C 180,E1 -14930.717,E2 -14930.717} C_VEL
LIN {X 0,Y 326.067,Z 667.869,A -85,B 0,C 180,E1 -14932.57,E2 -14932.57} C_VEL
LIN {X 0,Y 325.44,Z 670.035,A -85,B 0,C 180,E1 -14935.045,E2 -14935.045} C_VEL
LIN {X 0,Y 325.256,Z 670.761,A -85,B 0,C 180,E1 -14937.523,E2 -14937.523} C_VEL
LIN {X 0,Y 325.043,Z 670.061,A -85,B 0,C 180,E1 -14940,E2 -14940} C_VEL
LIN {X 0,Y 325.023,Z 667.91,A -85,B 0,C 180,E1 -14942.479,E2 -14942.479} C_VEL
LIN {X 0,Y 325.181,Z 664.253,A -85,B 0,C 180,E1 -14944.96,E2 -14944.96} C_VEL
LIN {X 0,Y 325.492,Z 658.932,A -85,B 0,C 180,E1 -14947.444,E2 -14947.444} C_VEL
LIN {X 0,Y 325.785,Z 653.818,A -85,B 0,C 180,E1 -14949.311,E2 -14949.311} C_VEL
LIN {X 0,Y 326.389,Z 646.391,A -85,B 0,C 180,E1 -14951.489,E2 -14951.489} C_VEL
LIN {X 0,Y 327.304,Z 637.2,A -85,B 0,C 180,E1 -14953.662,E2 -14953.662} C_VEL
LIN {X 0,Y 328.154,Z 627.931,A -85,B 0,C 180,E1 -14955.473,E2 -14955.473} C_VEL
LIN {X 0,Y 329.427,Z 616.107,A -85,B 0,C 180,E1 -14957.378,E2 -14957.378} C_VEL
LIN {X 0,Y 330.539,Z 604.486,A -85,B 0,C 180,E1 -14958.92,E2 -14958.92} C_VEL
LIN {X 0,Y 331.86,Z 591.873,A -85,B 0,C 180,E1 -14960.291,E2 -14960.291} C_VEL
LIN {X 0,Y 333.075,Z 577.948,A -85,B 0,C 180,E1 -14961.517,E2 -14961.517} C_VEL
LIN {X 0,Y 334.19,Z 562.696,A -85,B 0,C 180,E1 -14962.569,E2 -14962.569} C_VEL
LIN {X 0,Y 335.163,Z 547.135,A -85,B 0,C 180,E1 -14963.356,E2 -14963.356} C_VEL
LIN {X 0,Y 335.999,Z 528.413,A -85,B 0,C 180,E1 -14963.99,E2 -14963.99} C_VEL
LIN {X 0,Y 339.891,Z 435.01,A -85,B 0,C 180,E1 -14966.768,E2 -14966.768} C_VEL
LIN {X 0,Y 334.359,Z 398.118,A -85,B 0,C 180,E1 -14968.354,E2 -14968.354} C_VEL
LIN {X 0,Y 332.443,Z 388.878,A -85,B 0,C 180,E1 -14970.489,E2 -14970.489} C_VEL
LIN {X 0,Y 329.011,Z 374.169,A -85,B 0,C 180,E1 -14974.106,E2 -14974.106} C_VEL
LIN {X 0,Y 326.689,Z 364.75,A -85,B 0,C 180,E1 -14976.558,E2 -14976.558} C_VEL
LIN {X 0,Y 326.626,Z 364.427,A -85,B 0,C 180,E1 -14977.048,E2 -14977.048} C_VEL
LIN {X 0,Y 326.543,Z 364.425,A -85,B 0,C 180,E1 -14981.124,E2 -14981.124} C_VEL
LIN {X 0,Y 326.559,Z 364.413,A -85,B 0,C 180,E1 -14983.526,E2 -14983.526} C_VEL
LIN {X 0,Y 326.617,Z 364.507,A -85,B 0,C 180,E1 -14987.953,E2 -14987.953} C_VEL
LIN {X 0,Y 326.683,Z 365.006,A -85,B 0,C 180,E1 -14988.171,E2 -14988.171} C_VEL
LIN {X 0,Y 331.705,Z 379.383,A -85,B 0,C 180,E1 -14991.623,E2 -14991.623} C_VEL
LIN {X 0,Y 335.429,Z 391.965,A -85,B 0,C 180,E1 -14994.36,E2 -14994.36} C_VEL
LIN {X 0,Y 336.652,Z 396.257,A -85,B 0,C 180,E1 -14995.189,E2 -14995.189} C_VEL
LIN {X 0,Y 344.693,Z 413.874,A -85,B 0,C 180,E1 -14996.556,E2 -14996.556} C_VEL
LIN {X 0,Y 349.509,Z 440.842,A -85,B 0,C 180,E1 -14997.719,E2 -14997.719} C_VEL
LIN {X 0,Y 346.445,Z 542.36,A -85,B 0,C 180,E1 -14999.82,E2 -14999.82} C_VEL
LIN {X 0,Y 345.568,Z 566.859,A -85,B 0,C 180,E1 -15000.366,E2 -15000.366} C_VEL
LIN {X 0,Y 344.448,Z 582.358,A -85,B 0,C 180,E1 -15000.931,E2 -15000.931} C_VEL
LIN {X 0,Y 342.965,Z 597.252,A -85,B 0,C 180,E1 -15001.714,E2 -15001.714} C_VEL
LIN {X 0,Y 341.292,Z 610.985,A -85,B 0,C 180,E1 -15002.672,E2 -15002.672} C_VEL
LIN {X 0,Y 339.255,Z 624.753,A -85,B 0,C 180,E1 -15003.882,E2 -15003.882} C_VEL
LIN {X 0,Y 337.031,Z 638.157,A -85,B 0,C 180,E1 -15005.351,E2 -15005.351} C_VEL
LIN {X 0,Y 334.771,Z 650.326,A -85,B 0,C 180,E1 -15006.983,E2 -15006.983} C_VEL
LIN {X 0,Y 332.791,Z 661.131,A -85,B 0,C 180,E1 -15008.745,E2 -15008.745} C_VEL
LIN {X 0,Y 330.691,Z 671.493,A -85,B 0,C 180,E1 -15010.767,E2 -15010.767} C_VEL
LIN {X 0,Y 328.899,Z 680.558,A -85,B 0,C 180,E1 -15012.913,E2 -15012.913} C_VEL
LIN {X 0,Y 327.502,Z 688.087,A -85,B 0,C 180,E1 -15015.077,E2 -15015.077} C_VEL
LIN {X 0,Y 326.417,Z 695.11,A -85,B 0,C 180,E1 -15017.566,E2 -15017.566} C_VEL
LIN {X 0,Y 325.562,Z 700.635,A -85,B 0,C 180,E1 -15020.055,E2 -15020.055} C_VEL
LIN {X 0,Y 325.077,Z 704.817,A -85,B 0,C 180,E1 -15022.547,E2 -15022.547} C_VEL
LIN {X 0,Y 324.859,Z 707.755,A -85,B 0,C 180,E1 -15025.035,E2 -15025.035} C_VEL
LIN {X 0,Y 324.8,Z 709.516,A -85,B 0,C 180,E1 -15027.52,E2 -15027.52} C_VEL
LIN {X 0,Y 324.766,Z 710.125,A -85,B 0,C 180,E1 -15030,E2 -15030} C_VEL
LIN {X 0,Y 324.8,Z 709.554,A -85,B 0,C 180,E1 -15032.48,E2 -15032.48} C_VEL
LIN {X 0,Y 324.869,Z 707.844,A -85,B 0,C 180,E1 -15034.964,E2 -15034.964} C_VEL
LIN {X 0,Y 325.104,Z 704.965,A -85,B 0,C 180,E1 -15037.452,E2 -15037.452} C_VEL
LIN {X 0,Y 325.544,Z 700.847,A -85,B 0,C 180,E1 -15039.945,E2 -15039.945} C_VEL
LIN {X 0,Y 326.361,Z 695.379,A -85,B 0,C 180,E1 -15042.436,E2 -15042.436} C_VEL
LIN {X 0,Y 327.372,Z 689.088,A -85,B 0,C 180,E1 -15044.702,E2 -15044.702} C_VEL
LIN {X 0,Y 327.209,Z 686.309,A -85,B 0,C 180,E1 -15045.614,E2 -15045.614} C_VEL
LIN {X 0,Y 325.334,Z 681.572,A -85,B 0,C 180,E1 -15047.109,E2 -15047.109} C_VEL
LIN {X 0,Y 323.597,Z 676.44,A -85,B 0,C 180,E1 -15048.575,E2 -15048.575} C_VEL
LIN {X 0,Y 323.649,Z 672.967,A -85,B 0,C 180,E1 -15049.425,E2 -15049.425} C_VEL
LIN {X 0,Y 325.83,Z 662.784,A -85,B 0,C 180,E1 -15051.511,E2 -15051.511} C_VEL
LIN {X 0,Y 327.925,Z 651.94,A -85,B 0,C 180,E1 -15053.359,E2 -15053.359} C_VEL
LIN {X 0,Y 330.263,Z 640.09,A -85,B 0,C 180,E1 -15055.02,E2 -15055.02} C_VEL
LIN {X 0,Y 332.25,Z 628.51,A -85,B 0,C 180,E1 -15056.373,E2 -15056.373} C_VEL
LIN {X 0,Y 334.413,Z 615.106,A -85,B 0,C 180,E1 -15057.648,E2 -15057.648} C_VEL
LIN {X 0,Y 336.311,Z 600.869,A -85,B 0,C 180,E1 -15058.727,E2 -15058.727} C_VEL
LIN {X 0,Y 337.842,Z 586.466,A -85,B 0,C 180,E1 -15059.565,E2 -15059.565} C_VEL
LIN {X 0,Y 339.198,Z 570.78,A -85,B 0,C 180,E1 -15060.205,E2 -15060.205} C_VEL
LIN {X 0,Y 339.999,Z 554.024,A -85,B 0,C 180,E1 -15060.641,E2 -15060.641} C_VEL
LIN {X 0,Y 343.552,Z 441.944,A -85,B 0,C 180,E1 -15062.993,E2 -15062.993} C_VEL
LIN {X 0,Y 339.027,Z 416.699,A -85,B 0,C 180,E1 -15064.119,E2 -15064.119} C_VEL
LIN {X 0,Y 332.133,Z 401.531,A -85,B 0,C 180,E1 -15065.317,E2 -15065.317} C_VEL
LIN {X 0,Y 329.442,Z 395.851,A -85,B 0,C 180,E1 -15065.84,E2 -15065.84} C_VEL
LIN {X 0,Y 325.747,Z 383.414,A -85,B 0,C 180,E1 -15068.548,E2 -15068.548} C_VEL
LIN {X 0,Y 321.606,Z 371.185,A -85,B 0,C 180,E1 -15071.46,E2 -15071.46} C_VEL
LIN {X 0,Y 319.548,Z 365.458,A -85,B 0,C 180,E1 -15072.984,E2 -15072.984} C_VEL
LIN {X 0,Y 319.551,Z 365.304,A -85,B 0,C 180,E1 -15077.016,E2 -15077.016} C_VEL
LIN {X 0,Y 319.514,Z 365.304,A -85,B 0,C 180,E1 -15080.366,E2 -15080.366} C_VEL
LIN {X 0,Y 319.578,Z 365.29,A -85,B 0,C 180,E1 -15084.458,E2 -15084.458} C_VEL
LIN {X 0,Y 319.524,Z 365.295,A -85,B 0,C 180,E1 -15088.137,E2 -15088.137} C_VEL
LIN {X 0,Y 319.571,Z 365.295,A -85,B 0,C 180,E1 -15091.603,E2 -15091.603} C_VEL
LIN {X 0,Y 319.573,Z 365.304,A -85,B 0,C 180,E1 -15095.301,E2 -15095.301} C_VEL
LIN {X 0,Y 319.565,Z 365.285,A -85,B 0,C 180,E1 -15098.045,E2 -15098.045} C_VEL
LIN {X 0,Y 319.624,Z 365.284,A -85,B 0,C 180,E1 -15102.071,E2 -15102.071} C_VEL
LIN {X 0,Y 319.733,Z 365.283,A -85,B 0,C 180,E1 -15106.008,E2 -15106.008} C_VEL
LIN {X 0,Y 319.736,Z 365.263,A -85,B 0,C 180,E1 -15109.872,E2 -15109.872} C_VEL
LIN {X 0,Y 319.936,Z 365.245,A -85,B 0,C 180,E1 -15113.694,E2 -15113.694} C_VEL
LIN {X 0,Y 319.978,Z 365.248,A -85,B 0,C 180,E1 -15117.482,E2 -15117.482} C_VEL
LIN {X 0,Y 320.131,Z 365.222,A -85,B 0,C 180,E1 -15120,E2 -15120} C_VEL
LIN {X 0,Y 319.987,Z 365.233,A -85,B 0,C 180,E1 -15122.517,E2 -15122.517} C_VEL
LIN {X 0,Y 319.909,Z 365.248,A -85,B 0,C 180,E1 -15126.306,E2 -15126.306} C_VEL
LIN {X 0,Y 319.736,Z 365.279,A -85,B 0,C 180,E1 -15130.128,E2 -15130.128} C_VEL
LIN {X 0,Y 319.732,Z 365.258,A -85,B 0,C 180,E1 -15133.992,E2 -15133.992} C_VEL
LIN {X 0,Y 319.624,Z 365.289,A -85,B 0,C 180,E1 -15137.929,E2 -15137.929} C_VEL
LIN {X 0,Y 319.596,Z 365.3,A -85,B 0,C 180,E1 -15141.952,E2 -15141.952} C_VEL
LIN {X 0,Y 319.635,Z 365.284,A -85,B 0,C 180,E1 -15146.088,E2 -15146.088} C_VEL
LIN {X 0,Y 319.589,Z 365.29,A -85,B 0,C 180,E1 -15148.933,E2 -15148.933} C_VEL
LIN {X 0,Y 319.532,Z 365.309,A -85,B 0,C 180,E1 -15151.862,E2 -15151.862} C_VEL
LIN {X 0,Y 319.579,Z 365.295,A -85,B 0,C 180,E1 -15155.543,E2 -15155.543} C_VEL
LIN {X 0,Y 319.558,Z 365.254,A -85,B 0,C 180,E1 -15159.669,E2 -15159.669} C_VEL
LIN {X 0,Y 319.521,Z 365.311,A -85,B 0,C 180,E1 -15163.461,E2 -15163.461} C_VEL
LIN {X 0,Y 319.553,Z 365.265,A -85,B 0,C 180,E1 -15167.017,E2 -15167.017} C_VEL
LIN {X 0,Y 319.607,Z 365.552,A -85,B 0,C 180,E1 -15170.169,E2 -15170.169} C_VEL
LIN {X 0,Y 321.09,Z 371.025,A -85,B 0,C 180,E1 -15171.489,E2 -15171.489} C_VEL
LIN {X 0,Y 328.866,Z 391.984,A -85,B 0,C 180,E1 -15174.345,E2 -15174.345} C_VEL
LIN {X 0,Y 338.842,Z 413.946,A -85,B 0,C 180,E1 -15176.104,E2 -15176.104} C_VEL
LIN {X 0,Y 339.772,Z 416.956,A -85,B 0,C 180,E1 -15176.285,E2 -15176.285} C_VEL
LIN {X 0,Y 343.001,Z 439.321,A -85,B 0,C 180,E1 -15177.192,E2 -15177.192} C_VEL
LIN {X 0,Y 339.011,Z 563.854,A -85,B 0,C 180,E1 -15179.82,E2 -15179.82} C_VEL
LIN {X 0,Y 338.007,Z 578.689,A -85,B 0,C 180,E1 -15180.322,E2 -15180.322} C_VEL
LIN {X 0,Y 336.621,Z 593.281,A -85,B 0,C 180,E1 -15181.046,E2 -15181.046} C_VEL
LIN {X 0,Y 335.105,Z 606.246,A -85,B 0,C 180,E1 -15181.903,E2 -15181.903} C_VEL
LIN {X 0,Y 333.167,Z 619.781,A -85,B 0,C 180,E1 -15183.03,E2 -15183.03} C_VEL
LIN {X 0,Y 330.954,Z 632.72,A -85,B 0,C 180,E1 -15184.363,E2 -15184.363} C_VEL
LIN {X 0,Y 328.862,Z 644.637,A -85,B 0,C 180,E1 -15185.876,E2 -15185.876} C_VEL
LIN {X 0,Y 326.611,Z 656.181,A -85,B 0,C 180,E1 -15187.646,E2 -15187.646} C_VEL
LIN {X 0,Y 324.782,Z 665.778,A -85,B 0,C 180,E1 -15189.413,E2 -15189.413} C_VEL
LIN {X 0,Y 322.698,Z 675.653,A -85,B 0,C 180,E1 -15191.591,E2 -15191.591} C_VEL
LIN {X 0,Y 321.044,Z 683.84,A -85,B 0,C 180,E1 -15193.793,E2 -15193.793} C_VEL
LIN {X 0,Y 319.856,Z 690.609,A -85,B 0,C 180,E1 -15196.013,E2 -15196.013} C_VEL
LIN {X 0,Y 318.815,Z 696.876,A -85,B 0,C 180,E1 -15198.557,E2 -15198.557} C_VEL
LIN {X 0,Y 318.266,Z 701.71,A -85,B 0,C 180,E1 -15201.108,E2 -15201.108} C_VEL
LIN {X 0,Y 317.884,Z 705.243,A -85,B 0,C 180,E1 -15203.654,E2 -15203.654} C_VEL
LIN {X 0,Y 317.771,Z 707.567,A -85,B 0,C 180,E1 -15206.196,E2 -15206.196} C_VEL
LIN {X 0,Y 317.7,Z 708.735,A -85,B 0,C 180,E1 -15208.733,E2 -15208.733} C_VEL
LIN {X 0,Y 317.701,Z 708.733,A -85,B 0,C 180,E1 -15211.268,E2 -15211.268} C_VEL
LIN {X 0,Y 317.772,Z 707.56,A -85,B 0,C 180,E1 -15213.805,E2 -15213.805} C_VEL
LIN {X 0,Y 317.884,Z 705.228,A -85,B 0,C 180,E1 -15216.347,E2 -15216.347} C_VEL
LIN {X 0,Y 318.266,Z 701.679,A -85,B 0,C 180,E1 -15218.892,E2 -15218.892} C_VEL
LIN {X 0,Y 318.818,Z 696.833,A -85,B 0,C 180,E1 -15221.443,E2 -15221.443} C_VEL
LIN {X 0,Y 319.858,Z 690.562,A -85,B 0,C 180,E1 -15223.987,E2 -15223.987} C_VEL
LIN {X 0,Y 321.307,Z 682.672,A -85,B 0,C 180,E1 -15226.52,E2 -15226.52} C_VEL
LIN {X 0,Y 322.966,Z 674.24,A -85,B 0,C 180,E1 -15228.722,E2 -15228.722} C_VEL
LIN {X 0,Y 324.765,Z 665.686,A -85,B 0,C 180,E1 -15230.589,E2 -15230.589} C_VEL
LIN {X 0,Y 326.814,Z 655.27,A -85,B 0,C 180,E1 -15232.49,E2 -15232.49} C_VEL
LIN {X 0,Y 331.477,Z 633.378,A -85,B 0,C 180,E1 -15235.763,E2 -15235.763} C_VEL
LIN {X 0,Y 334.496,Z 620.487,A -85,B 0,C 180,E1 -15237.362,E2 -15237.362} C_VEL
LIN {X 0,Y 337.635,Z 605.908,A -85,B 0,C 180,E1 -15238.841,E2 -15238.841} C_VEL
LIN {X 0,Y 340.569,Z 591.169,A -85,B 0,C 180,E1 -15240.028,E2 -15240.028} C_VEL
LIN {X 0,Y 343.172,Z 576.356,A -85,B 0,C 180,E1 -15240.967,E2 -15240.967} C_VEL
LIN {X 0,Y 345.474,Z 560.85,A -85,B 0,C 180,E1 -15241.718,E2 -15241.718} C_VEL
LIN {X 0,Y 355.58,Z 474.523,A -85,B 0,C 180,E1 -15244.757,E2 -15244.757} C_VEL
LIN {X 0,Y 359.76,Z 442.731,A -85,B 0,C 180,E1 -15245.916,E2 -15245.916} C_VEL
LIN {X 0,Y 359.571,Z 438.345,A -85,B 0,C 180,E1 -15246.298,E2 -15246.298} C_VEL
LIN {X 0,Y 356.899,Z 432.172,A -85,B 0,C 180,E1 -15247.644,E2 -15247.644} C_VEL
LIN {X 0,Y 354.964,Z 428.245,A -85,B 0,C 180,E1 -15248.736,E2 -15248.736} C_VEL
LIN {X 0,Y 352.746,Z 424.045,A -85,B 0,C 180,E1 -15250.217,E2 -15250.217} C_VEL
LIN {X 0,Y 350.124,Z 419.642,A -85,B 0,C 180,E1 -15252.624,E2 -15252.624} C_VEL
LIN {X 0,Y 348.826,Z 418.028,A -85,B 0,C 180,E1 -15254.661,E2 -15254.661} C_VEL
LIN {X 0,Y 348.469,Z 417.751,A -85,B 0,C 180,E1 -15256.708,E2 -15256.708} C_VEL
LIN {X 0,Y 349.117,Z 418.677,A -85,B 0,C 180,E1 -15258.78,E2 -15258.78} C_VEL
LIN {X 0,Y 350.145,Z 420.353,A -85,B 0,C 180,E1 -15260.271,E2 -15260.271} C_VEL
LIN {X 0,Y 352.72,Z 425.131,A -85,B 0,C 180,E1 -15262.67,E2 -15262.67} C_VEL
LIN {X 0,Y 355.239,Z 430.489,A -85,B 0,C 180,E1 -15264.386,E2 -15264.386} C_VEL
LIN {X 0,Y 357.223,Z 435.214,A -85,B 0,C 180,E1 -15265.549,E2 -15265.549} C_VEL
LIN {X 0,Y 358.61,Z 439.022,A -85,B 0,C 180,E1 -15266.312,E2 -15266.312} C_VEL
LIN {X 0,Y 359.025,Z 447.083,A -85,B 0,C 180,E1 -15267.083,E2 -15267.083} C_VEL
LIN {X 0,Y 348.018,Z 527.989,A -85,B 0,C 180,E1 -15270.18,E2 -15270.18} C_VEL
LIN {X 0,Y 344.902,Z 553.115,A -85,B 0,C 180,E1 -15271.222,E2 -15271.222} C_VEL
LIN {X 0,Y 342.312,Z 569.666,A -85,B 0,C 180,E1 -15272.195,E2 -15272.195} C_VEL
LIN {X 0,Y 339.519,Z 585.481,A -85,B 0,C 180,E1 -15273.437,E2 -15273.437} C_VEL
LIN {X 0,Y 336.598,Z 599.506,A -85,B 0,C 180,E1 -15274.823,E2 -15274.823} C_VEL
LIN {X 0,Y 333.658,Z 612.474,A -85,B 0,C 180,E1 -15276.409,E2 -15276.409} C_VEL
LIN {X 0,Y 330.872,Z 624.235,A -85,B 0,C 180,E1 -15278.179,E2 -15278.179} C_VEL
LIN {X 0,Y 328.434,Z 634.071,A -85,B 0,C 180,E1 -15279.978,E2 -15279.978} C_VEL
LIN {X 0,Y 325.889,Z 643.314,A -85,B 0,C 180,E1 -15282.016,E2 -15282.016} C_VEL
LIN {X 0,Y 323.69,Z 651.455,A -85,B 0,C 180,E1 -15284.252,E2 -15284.252} C_VEL
LIN {X 0,Y 322.221,Z 656.995,A -85,B 0,C 180,E1 -15286.118,E2 -15286.118} C_VEL
LIN {X 0,Y 321.02,Z 661.5,A -85,B 0,C 180,E1 -15287.996,E2 -15287.996} C_VEL
LIN {X 0,Y 320.104,Z 665.087,A -85,B 0,C 180,E1 -15289.884,E2 -15289.884} C_VEL
LIN {X 0,Y 319.06,Z 668.568,A -85,B 0,C 180,E1 -15292.406,E2 -15292.406} C_VEL
LIN {X 0,Y 318.39,Z 670.589,A -85,B 0,C 180,E1 -15294.935,E2 -15294.935} C_VEL
LIN {X 0,Y 318.17,Z 671.172,A -85,B 0,C 180,E1 -15297.468,E2 -15297.468} C_VEL
LIN {X 0,Y 317.948,Z 670.334,A -85,B 0,C 180,E1 -15300,E2 -15300} C_VEL
LIN {X 0,Y 317.938,Z 668.036,A -85,B 0,C 180,E1 -15302.534,E2 -15302.534} C_VEL
LIN {X 0,Y 318.035,Z 665.283,A -85,B 0,C 180,E1 -15304.436,E2 -15304.436} C_VEL
LIN {X 0,Y 318.322,Z 660.264,A -85,B 0,C 180,E1 -15306.975,E2 -15306.975} C_VEL
LIN {X 0,Y 318.59,Z 655.32,A -85,B 0,C 180,E1 -15308.883,E2 -15308.883} C_VEL
LIN {X 0,Y 319.197,Z 648.203,A -85,B 0,C 180,E1 -15311.108,E2 -15311.108} C_VEL
LIN {X 0,Y 320.055,Z 639.377,A -85,B 0,C 180,E1 -15313.331,E2 -15313.331} C_VEL
LIN {X 0,Y 321.013,Z 629.175,A -85,B 0,C 180,E1 -15315.412,E2 -15315.412} C_VEL
LIN {X 0,Y 322.222,Z 617.986,A -85,B 0,C 180,E1 -15317.288,E2 -15317.288} C_VEL
LIN {X 0,Y 323.475,Z 605.459,A -85,B 0,C 180,E1 -15319.02,E2 -15319.02} C_VEL
LIN {X 0,Y 324.79,Z 593.048,A -85,B 0,C 180,E1 -15320.422,E2 -15320.422} C_VEL
LIN {X 0,Y 326.087,Z 579.006,A -85,B 0,C 180,E1 -15321.701,E2 -15321.701} C_VEL
LIN {X 0,Y 327.156,Z 564.459,A -85,B 0,C 180,E1 -15322.748,E2 -15322.748} C_VEL
LIN {X 0,Y 328.205,Z 548.882,A -85,B 0,C 180,E1 -15323.589,E2 -15323.589} C_VEL
LIN {X 0,Y 328.995,Z 532.135,A -85,B 0,C 180,E1 -15324.198,E2 -15324.198} C_VEL
LIN {X 0,Y 333.158,Z 435.714,A -85,B 0,C 180,E1 -15327.154,E2 -15327.154} C_VEL
LIN {X 0,Y 327.778,Z 399.859,A -85,B 0,C 180,E1 -15328.714,E2 -15328.714} C_VEL
LIN {X 0,Y 327.191,Z 397.693,A -85,B 0,C 180,E1 -15328.912,E2 -15328.912} C_VEL
LIN {X 0,Y 323.873,Z 383.178,A -85,B 0,C 180,E1 -15332.446,E2 -15332.446} C_VEL
LIN {X 0,Y 320.742,Z 369.993,A -85,B 0,C 180,E1 -15335.832,E2 -15335.832} C_VEL
LIN {X 0,Y 319.602,Z 365.449,A -85,B 0,C 180,E1 -15337.11,E2 -15337.11} C_VEL
LIN {X 0,Y 319.498,Z 365.298,A -85,B 0,C 180,E1 -15341.293,E2 -15341.293} C_VEL
LIN {X 0,Y 319.519,Z 365.288,A -85,B 0,C 180,E1 -15343.46,E2 -15343.46} C_VEL
LIN {X 0,Y 319.576,Z 365.506,A -85,B 0,C 180,E1 -15347.172,E2 -15347.172} C_VEL
LIN {X 0,Y 324.726,Z 380.285,A -85,B 0,C 180,E1 -15350.857,E2 -15350.857} C_VEL
LIN {X 0,Y 328.764,Z 393.513,A -85,B 0,C 180,E1 -15353.802,E2 -15353.802} C_VEL
LIN {X 0,Y 329.717,Z 396.593,A -85,B 0,C 180,E1 -15354.368,E2 -15354.368} C_VEL
LIN {X 0,Y 337.427,Z 413.107,A -85,B 0,C 180,E1 -15355.721,E2 -15355.721} C_VEL
LIN {X 0,Y 339.328,Z 417.968,A -85,B 0,C 180,E1 -15356.06,E2 -15356.06} C_VEL
LIN {X 0,Y 343.438,Z 441.536,A -85,B 0,C 180,E1 -15357.097,E2 -15357.097} C_VEL
LIN {X 0,Y 340.961,Z 523.34,A -85,B 0,C 180,E1 -15358.826,E2 -15358.826} C_VEL
LIN {X 0,Y 339.486,Z 565.411,A -85,B 0,C 180,E1 -15359.737,E2 -15359.737} C_VEL
LIN {X 0,Y 338.377,Z 580.581,A -85,B 0,C 180,E1 -15360.272,E2 -15360.272} C_VEL
LIN {X 0,Y 336.952,Z 594.719,A -85,B 0,C 180,E1 -15360.991,E2 -15360.991} C_VEL
LIN {X 0,Y 335.202,Z 608.799,A -85,B 0,C 180,E1 -15361.943,E2 -15361.943} C_VEL
LIN {X 0,Y 333.377,Z 621.642,A -85,B 0,C 180,E1 -15363.048,E2 -15363.048} C_VEL
LIN {X 0,Y 331.22,Z 634.342,A -85,B 0,C 180,E1 -15364.384,E2 -15364.384} C_VEL
LIN {X 0,Y 328.84,Z 647.155,A -85,B 0,C 180,E1 -15366.042,E2 -15366.042} C_VEL
LIN {X 0,Y 326.803,Z 657.373,A -85,B 0,C 180,E1 -15367.628,E2 -15367.628} C_VEL
LIN {X 0,Y 324.945,Z 667.065,A -85,B 0,C 180,E1 -15369.423,E2 -15369.423} C_VEL
LIN {X 0,Y 322.854,Z 676.884,A -85,B 0,C 180,E1 -15371.6,E2 -15371.6} C_VEL
LIN {X 0,Y 321.19,Z 685.146,A -85,B 0,C 180,E1 -15373.833,E2 -15373.833} C_VEL
LIN {X 0,Y 319.95,Z 691.784,A -85,B 0,C 180,E1 -15376.017,E2 -15376.017} C_VEL
LIN {X 0,Y 318.869,Z 698.035,A -85,B 0,C 180,E1 -15378.559,E2 -15378.559} C_VEL
LIN {X 0,Y 318.274,Z 702.873,A -85,B 0,C 180,E1 -15381.108,E2 -15381.108} C_VEL
LIN {X 0,Y 317.882,Z 706.423,A -85,B 0,C 180,E1 -15383.653,E2 -15383.653} C_VEL
LIN {X 0,Y 317.758,Z 708.766,A -85,B 0,C 180,E1 -15386.195,E2 -15386.195} C_VEL
LIN {X 0,Y 317.688,Z 709.955,A -85,B 0,C 180,E1 -15388.732,E2 -15388.732} C_VEL
LIN {X 0,Y 317.688,Z 709.968,A -85,B 0,C 180,E1 -15391.267,E2 -15391.267} C_VEL
LIN {X 0,Y 317.761,Z 708.828,A -85,B 0,C 180,E1 -15393.804,E2 -15393.804} C_VEL
LIN {X 0,Y 317.885,Z 706.539,A -85,B 0,C 180,E1 -15396.346,E2 -15396.346} C_VEL
LIN {X 0,Y 318.271,Z 703.051,A -85,B 0,C 180,E1 -15398.892,E2 -15398.892} C_VEL
LIN {X 0,Y 318.841,Z 698.274,A -85,B 0,C 180,E1 -15401.442,E2 -15401.442} C_VEL
LIN {X 0,Y 319.918,Z 692.079,A -85,B 0,C 180,E1 -15403.984,E2 -15403.984} C_VEL
LIN {X 0,Y 321.355,Z 684.293,A -85,B 0,C 180,E1 -15406.517,E2 -15406.517} C_VEL
LIN {X 0,Y 323.035,Z 675.995,A -85,B 0,C 180,E1 -15408.717,E2 -15408.717} C_VEL
LIN {X 0,Y 323.649,Z 672.967,A -85,B 0,C 180,E1 -15409.425,E2 -15409.425} C_VEL
LIN {X 0,Y 323.74,Z 669.385,A -85,B 0,C 180,E1 -15410.258,E2 -15410.258} C_VEL
LIN {X 0,Y 322.265,Z 663.408,A -85,B 0,C 180,E1 -15411.639,E2 -15411.639} C_VEL
LIN {X 0,Y 320.915,Z 657.08,A -85,B 0,C 180,E1 -15412.97,E2 -15412.97} C_VEL
LIN {X 0,Y 321.184,Z 652.854,A -85,B 0,C 180,E1 -15413.711,E2 -15413.711} C_VEL
LIN {X 0,Y 323.591,Z 641.214,A -85,B 0,C 180,E1 -15415.401,E2 -15415.401} C_VEL
LIN {X 0,Y 325.883,Z 628.478,A -85,B 0,C 180,E1 -15416.929,E2 -15416.929} C_VEL
LIN {X 0,Y 327.962,Z 616.169,A -85,B 0,C 180,E1 -15418.128,E2 -15418.128} C_VEL
LIN {X 0,Y 329.951,Z 602.026,A -85,B 0,C 180,E1 -15419.237,E2 -15419.237} C_VEL
LIN {X 0,Y 331.619,Z 587.132,A -85,B 0,C 180,E1 -15420.133,E2 -15420.133} C_VEL
LIN {X 0,Y 333,Z 571.755,A -85,B 0,C 180,E1 -15420.784,E2 -15420.784} C_VEL
LIN {X 0,Y 333.92,Z 553.872,A -85,B 0,C 180,E1 -15421.261,E2 -15421.261} C_VEL
LIN {X 0,Y 337.579,Z 443.242,A -85,B 0,C 180,E1 -15423.617,E2 -15423.617} C_VEL
LIN {X 0,Y 333.394,Z 419.51,A -85,B 0,C 180,E1 -15424.701,E2 -15424.701} C_VEL
LIN {X 0,Y 326.101,Z 403.481,A -85,B 0,C 180,E1 -15426.015,E2 -15426.015} C_VEL
LIN {X 0,Y 322.337,Z 395.811,A -85,B 0,C 180,E1 -15426.749,E2 -15426.749} C_VEL
LIN {X 0,Y 318.643,Z 383.729,A -85,B 0,C 180,E1 -15429.469,E2 -15429.469} C_VEL
LIN {X 0,Y 314.42,Z 371.625,A -85,B 0,C 180,E1 -15432.47,E2 -15432.47} C_VEL
LIN {X 0,Y 312.474,Z 366.396,A -85,B 0,C 180,E1 -15433.91,E2 -15433.91} C_VEL
LIN {X 0,Y 312.465,Z 366.183,A -85,B 0,C 180,E1 -15437.564,E2 -15437.564} C_VEL
LIN {X 0,Y 312.455,Z 366.181,A -85,B 0,C 180,E1 -15440.964,E2 -15440.964} C_VEL
LIN {X 0,Y 312.529,Z 366.168,A -85,B 0,C 180,E1 -15444.22,E2 -15444.22} C_VEL
LIN {X 0,Y 312.501,Z 366.176,A -85,B 0,C 180,E1 -15447.333,E2 -15447.333} C_VEL
LIN {X 0,Y 312.506,Z 366.179,A -85,B 0,C 180,E1 -15451.292,E2 -15451.292} C_VEL
LIN {X 0,Y 312.547,Z 366.176,A -85,B 0,C 180,E1 -15454.707,E2 -15454.707} C_VEL
LIN {X 0,Y 312.526,Z 366.168,A -85,B 0,C 180,E1 -15458.912,E2 -15458.912} C_VEL
LIN {X 0,Y 312.582,Z 366.164,A -85,B 0,C 180,E1 -15461.653,E2 -15461.653} C_VEL
LIN {X 0,Y 312.686,Z 366.161,A -85,B 0,C 180,E1 -15465.686,E2 -15465.686} C_VEL
LIN {X 0,Y 312.686,Z 366.139,A -85,B 0,C 180,E1 -15469.641,E2 -15469.641} C_VEL
LIN {X 0,Y 312.892,Z 366.123,A -85,B 0,C 180,E1 -15473.552,E2 -15473.552} C_VEL
LIN {X 0,Y 312.987,Z 366.123,A -85,B 0,C 180,E1 -15478.713,E2 -15478.713} C_VEL
LIN {X 0,Y 312.987,Z 366.098,A -85,B 0,C 180,E1 -15481.287,E2 -15481.287} C_VEL
LIN {X 0,Y 312.704,Z 366.157,A -85,B 0,C 180,E1 -15485.158,E2 -15485.158} C_VEL
LIN {X 0,Y 312.802,Z 366.12,A -85,B 0,C 180,E1 -15487.747,E2 -15487.747} C_VEL
LIN {X 0,Y 312.664,Z 366.157,A -85,B 0,C 180,E1 -15491.671,E2 -15491.671} C_VEL
LIN {X 0,Y 312.668,Z 366.144,A -85,B 0,C 180,E1 -15494.865,E2 -15494.865} C_VEL
LIN {X 0,Y 312.586,Z 366.152,A -85,B 0,C 180,E1 -15499.213,E2 -15499.213} C_VEL
LIN {X 0,Y 312.546,Z 366.179,A -85,B 0,C 180,E1 -15502.789,E2 -15502.789} C_VEL
LIN {X 0,Y 312.603,Z 366.158,A -85,B 0,C 180,E1 -15505.936,E2 -15505.936} C_VEL
LIN {X 0,Y 312.545,Z 366.161,A -85,B 0,C 180,E1 -15509.65,E2 -15509.65} C_VEL
LIN {X 0,Y 312.519,Z 366.17,A -85,B 0,C 180,E1 -15513.689,E2 -15513.689} C_VEL
LIN {X 0,Y 312.52,Z 366.174,A -85,B 0,C 180,E1 -15517.386,E2 -15517.386} C_VEL
LIN {X 0,Y 312.489,Z 366.133,A -85,B 0,C 180,E1 -15520.709,E2 -15520.709} C_VEL
LIN {X 0,Y 312.451,Z 366.186,A -85,B 0,C 180,E1 -15524.21,E2 -15524.21} C_VEL
LIN {X 0,Y 312.483,Z 366.152,A -85,B 0,C 180,E1 -15527.919,E2 -15527.919} C_VEL
LIN {X 0,Y 312.554,Z 366.409,A -85,B 0,C 180,E1 -15529.611,E2 -15529.611} C_VEL
LIN {X 0,Y 313.039,Z 368.089,A -85,B 0,C 180,E1 -15530,E2 -15530} C_VEL
LIN {X 0,Y 320.788,Z 388.719,A -85,B 0,C 180,E1 -15533.027,E2 -15533.027} C_VEL
LIN {X 0,Y 322.254,Z 392.657,A -85,B 0,C 180,E1 -15533.511,E2 -15533.511} C_VEL
LIN {X 0,Y 332.247,Z 414.584,A -85,B 0,C 180,E1 -15535.348,E2 -15535.348} C_VEL
LIN {X 0,Y 334.062,Z 419.362,A -85,B 0,C 180,E1 -15535.686,E2 -15535.686} C_VEL
LIN {X 0,Y 336.997,Z 439.462,A -85,B 0,C 180,E1 -15536.532,E2 -15536.532} C_VEL
LIN {X 0,Y 333.147,Z 559.607,A -85,B 0,C 180,E1 -15539.1,E2 -15539.1} C_VEL
LIN {X 0,Y 332.159,Z 575.172,A -85,B 0,C 180,E1 -15539.57,E2 -15539.57} C_VEL
LIN {X 0,Y 330.85,Z 589.492,A -85,B 0,C 180,E1 -15540.229,E2 -15540.229} C_VEL
LIN {X 0,Y 329.229,Z 603.063,A -85,B 0,C 180,E1 -15541.071,E2 -15541.071} C_VEL
LIN {X 0,Y 327.388,Z 616.612,A -85,B 0,C 180,E1 -15542.167,E2 -15542.167} C_VEL
LIN {X 0,Y 325.071,Z 630.135,A -85,B 0,C 180,E1 -15543.519,E2 -15543.519} C_VEL
LIN {X 0,Y 322.793,Z 642.465,A -85,B 0,C 180,E1 -15545.049,E2 -15545.049} C_VEL
LIN {X 0,Y 320.499,Z 653.789,A -85,B 0,C 180,E1 -15546.752,E2 -15546.752} C_VEL
LIN {X 0,Y 318.429,Z 664.187,A -85,B 0,C 180,E1 -15548.644,E2 -15548.644} C_VEL
LIN {X 0,Y 316.475,Z 672.992,A -85,B 0,C 180,E1 -15550.543,E2 -15550.543} C_VEL
LIN {X 0,Y 314.655,Z 681.638,A -85,B 0,C 180,E1 -15552.786,E2 -15552.786} C_VEL
LIN {X 0,Y 313.142,Z 689.472,A -85,B 0,C 180,E1 -15555.282,E2 -15555.282} C_VEL
LIN {X 0,Y 312.081,Z 695.474,A -85,B 0,C 180,E1 -15557.647,E2 -15557.647} C_VEL
LIN {X 0,Y 311.315,Z 700.666,A -85,B 0,C 180,E1 -15560.252,E2 -15560.252} C_VEL
LIN {X 0,Y 310.967,Z 703.647,A -85,B 0,C 180,E1 -15562.207,E2 -15562.207} C_VEL
LIN {X 0,Y 310.691,Z 706.566,A -85,B 0,C 180,E1 -15564.809,E2 -15564.809} C_VEL
LIN {X 0,Y 310.674,Z 708.307,A -85,B 0,C 180,E1 -15567.407,E2 -15567.407} C_VEL
LIN {X 0,Y 310.592,Z 708.9,A -85,B 0,C 180,E1 -15570,E2 -15570} C_VEL
LIN {X 0,Y 310.675,Z 708.303,A -85,B 0,C 180,E1 -15572.593,E2 -15572.593} C_VEL
LIN {X 0,Y 310.691,Z 706.555,A -85,B 0,C 180,E1 -15575.192,E2 -15575.192} C_VEL
LIN {X 0,Y 310.967,Z 703.623,A -85,B 0,C 180,E1 -15577.794,E2 -15577.794} C_VEL
LIN {X 0,Y 311.465,Z 699.439,A -85,B 0,C 180,E1 -15580.4,E2 -15580.4} C_VEL
LIN {X 0,Y 312.37,Z 693.9,A -85,B 0,C 180,E1 -15583.002,E2 -15583.002} C_VEL
LIN {X 0,Y 313.599,Z 686.849,A -85,B 0,C 180,E1 -15585.601,E2 -15585.601} C_VEL
LIN {X 0,Y 315.149,Z 679.28,A -85,B 0,C 180,E1 -15587.857,E2 -15587.857} C_VEL
LIN {X 0,Y 317.049,Z 670.151,A -85,B 0,C 180,E1 -15590.096,E2 -15590.096} C_VEL
LIN {X 0,Y 319.099,Z 660.85,A -85,B 0,C 180,E1 -15591.989,E2 -15591.989} C_VEL
LIN {X 0,Y 323.754,Z 640.977,A -85,B 0,C 180,E1 -15595.387,E2 -15595.387} C_VEL
LIN {X 0,Y 326.962,Z 628.462,A -85,B 0,C 180,E1 -15597.179,E2 -15597.179} C_VEL
LIN {X 0,Y 330.277,Z 614.845,A -85,B 0,C 180,E1 -15598.78,E2 -15598.78} C_VEL
LIN {X 0,Y 333.402,Z 601.01,A -85,B 0,C 180,E1 -15600.104,E2 -15600.104} C_VEL
LIN {X 0,Y 336.577,Z 585.648,A -85,B 0,C 180,E1 -15601.275,E2 -15601.275} C_VEL
LIN {X 0,Y 339.407,Z 570.068,A -85,B 0,C 180,E1 -15602.178,E2 -15602.178} C_VEL
LIN {X 0,Y 341.656,Z 554.634,A -85,B 0,C 180,E1 -15602.857,E2 -15602.857} C_VEL
LIN {X 0,Y 349.829,Z 488.463,A -85,B 0,C 180,E1 -15605.237,E2 -15605.237} C_VEL
LIN {X 0,Y 356.073,Z 444.488,A -85,B 0,C 180,E1 -15606.853,E2 -15606.853} C_VEL
LIN {X 0,Y 355.946,Z 442.522,A -85,B 0,C 180,E1 -15607.058,E2 -15607.058} C_VEL
LIN {X 0,Y 353.81,Z 437.466,A -85,B 0,C 180,E1 -15608.248,E2 -15608.248} C_VEL
LIN {X 0,Y 352.249,Z 434.112,A -85,B 0,C 180,E1 -15609.225,E2 -15609.225} C_VEL
LIN {X 0,Y 350.41,Z 430.393,A -85,B 0,C 180,E1 -15610.578,E2 -15610.578} C_VEL
LIN {X 0,Y 348.159,Z 426.373,A -85,B 0,C 180,E1 -15612.819,E2 -15612.819} C_VEL
LIN {X 0,Y 347.085,Z 424.944,A -85,B 0,C 180,E1 -15614.579,E2 -15614.579} C_VEL
LIN {X 0,Y 346.706,Z 424.649,A -85,B 0,C 180,E1 -15616.866,E2 -15616.866} C_VEL
LIN {X 0,Y 347.407,Z 425.692,A -85,B 0,C 180,E1 -15618.942,E2 -15618.942} C_VEL
LIN {X 0,Y 348.317,Z 427.51,A -85,B 0,C 180,E1 -15620.326,E2 -15620.326} C_VEL
LIN {X 0,Y 350.404,Z 431.626,A -85,B 0,C 180,E1 -15622.376,E2 -15622.376} C_VEL
LIN {X 0,Y 352.561,Z 436.648,A -85,B 0,C 180,E1 -15624.001,E2 -15624.001} C_VEL
LIN {X 0,Y 354.659,Z 441.999,A -85,B 0,C 180,E1 -15625.325,E2 -15625.325} C_VEL
LIN {X 0,Y 355.105,Z 443.796,A -85,B 0,C 180,E1 -15625.642,E2 -15625.642} C_VEL
LIN {X 0,Y 355.202,Z 449.183,A -85,B 0,C 180,E1 -15626.157,E2 -15626.157} C_VEL
LIN {X 0,Y 343.139,Z 532.279,A -85,B 0,C 180,E1 -15629.414,E2 -15629.414} C_VEL
LIN {X 0,Y 340.102,Z 554.63,A -85,B 0,C 180,E1 -15630.381,E2 -15630.381} C_VEL
LIN {X 0,Y 337.317,Z 570.807,A -85,B 0,C 180,E1 -15631.367,E2 -15631.367} C_VEL
LIN {X 0,Y 334.35,Z 586.358,A -85,B 0,C 180,E1 -15632.625,E2 -15632.625} C_VEL
LIN {X 0,Y 331.486,Z 599.111,A -85,B 0,C 180,E1 -15633.901,E2 -15633.901} C_VEL
LIN {X 0,Y 328.608,Z 611.012,A -85,B 0,C 180,E1 -15635.352,E2 -15635.352} C_VEL
LIN {X 0,Y 325.535,Z 622.97,A -85,B 0,C 180,E1 -15637.133,E2 -15637.133} C_VEL
LIN {X 0,Y 322.865,Z 633.001,A -85,B 0,C 180,E1 -15638.951,E2 -15638.951} C_VEL
LIN {X 0,Y 320.391,Z 641.511,A -85,B 0,C 180,E1 -15640.79,E2 -15640.79} C_VEL
LIN {X 0,Y 318.255,Z 648.693,A -85,B 0,C 180,E1 -15642.655,E2 -15642.655} C_VEL
LIN {X 0,Y 316.437,Z 654.736,A -85,B 0,C 180,E1 -15644.543,E2 -15644.543} C_VEL
LIN {X 0,Y 314.447,Z 661.184,A -85,B 0,C 180,E1 -15647.085,E2 -15647.085} C_VEL
LIN {X 0,Y 313.183,Z 665.971,A -85,B 0,C 180,E1 -15649.658,E2 -15649.658} C_VEL
LIN {X 0,Y 312.02,Z 669.398,A -85,B 0,C 180,E1 -15652.337,E2 -15652.337} C_VEL
LIN {X 0,Y 311.344,Z 671.154,A -85,B 0,C 180,E1 -15654.82,E2 -15654.82} C_VEL
LIN {X 0,Y 311.084,Z 671.584,A -85,B 0,C 180,E1 -15657.41,E2 -15657.41} C_VEL
LIN {X 0,Y 310.853,Z 670.576,A -85,B 0,C 180,E1 -15660,E2 -15660} C_VEL
LIN {X 0,Y 310.855,Z 668.099,A -85,B 0,C 180,E1 -15662.592,E2 -15662.592} C_VEL
LIN {X 0,Y 310.958,Z 665.26,A -85,B 0,C 180,E1 -15664.537,E2 -15664.537} C_VEL
LIN {X 0,Y 311.25,Z 660.052,A -85,B 0,C 180,E1 -15667.134,E2 -15667.134} C_VEL
LIN {X 0,Y 311.529,Z 654.989,A -85,B 0,C 180,E1 -15669.086,E2 -15669.086} C_VEL
LIN {X 0,Y 312.151,Z 647.678,A -85,B 0,C 180,E1 -15671.362,E2 -15671.362} C_VEL
LIN {X 0,Y 313.097,Z 638.586,A -85,B 0,C 180,E1 -15673.632,E2 -15673.632} C_VEL
LIN {X 0,Y 314,Z 629.125,A -85,B 0,C 180,E1 -15675.58,E2 -15675.58} C_VEL
LIN {X 0,Y 315.248,Z 617.755,A -85,B 0,C 180,E1 -15677.516,E2 -15677.516} C_VEL
LIN {X 0,Y 316.522,Z 605.121,A -85,B 0,C 180,E1 -15679.286,E2 -15679.286} C_VEL
LIN {X 0,Y 317.905,Z 592.569,A -85,B 0,C 180,E1 -15680.715,E2 -15680.715} C_VEL
LIN {X 0,Y 319.184,Z 578.845,A -85,B 0,C 180,E1 -15681.982,E2 -15681.982} C_VEL
LIN {X 0,Y 320.253,Z 564.687,A -85,B 0,C 180,E1 -15683.021,E2 -15683.021} C_VEL
LIN {X 0,Y 321.298,Z 549.343,A -85,B 0,C 180,E1 -15683.87,E2 -15683.87} C_VEL
LIN {X 0,Y 322.115,Z 532.948,A -85,B 0,C 180,E1 -15684.491,E2 -15684.491} C_VEL
LIN {X 0,Y 326.463,Z 436.599,A -85,B 0,C 180,E1 -15687.542,E2 -15687.542} C_VEL
LIN {X 0,Y 321.097,Z 401.271,A -85,B 0,C 180,E1 -15689.126,E2 -15689.126} C_VEL
LIN {X 0,Y 319.995,Z 397.941,A -85,B 0,C 180,E1 -15689.368,E2 -15689.368} C_VEL
LIN {X 0,Y 316.623,Z 383.098,A -85,B 0,C 180,E1 -15693.061,E2 -15693.061} C_VEL
LIN {X 0,Y 313.412,Z 369.812,A -85,B 0,C 180,E1 -15696.559,E2 -15696.559} C_VEL
LIN {X 0,Y 312.529,Z 366.376,A -85,B 0,C 180,E1 -15697.555,E2 -15697.555} C_VEL
LIN {X 0,Y 312.441,Z 366.188,A -85,B 0,C 180,E1 -15700.717,E2 -15700.717} C_VEL
LIN {X 0,Y 312.451,Z 366.178,A -85,B 0,C 180,E1 -15704.21,E2 -15704.21} C_VEL
LIN {X 0,Y 312.497,Z 366.399,A -85,B 0,C 180,E1 -15706.231,E2 -15706.231} C_VEL
LIN {X 0,Y 316.989,Z 378.928,A -85,B 0,C 180,E1 -15709.49,E2 -15709.49} C_VEL
LIN {X 0,Y 320.229,Z 388.802,A -85,B 0,C 180,E1 -15711.839,E2 -15711.839} C_VEL
LIN {X 0,Y 322.596,Z 396.464,A -85,B 0,C 180,E1 -15713.456,E2 -15713.456} C_VEL
LIN {X 0,Y 330.498,Z 412.973,A -85,B 0,C 180,E1 -15714.898,E2 -15714.898} C_VEL
LIN {X 0,Y 333.581,Z 420.124,A -85,B 0,C 180,E1 -15715.451,E2 -15715.451} C_VEL
LIN {X 0,Y 337.519,Z 443.829,A -85,B 0,C 180,E1 -15716.504,E2 -15716.504} C_VEL
LIN {X 0,Y 333.883,Z 552.854,A -85,B 0,C 180,E1 -15718.823,E2 -15718.823} C_VEL
LIN {X 0,Y 333.082,Z 570.071,A -85,B 0,C 180,E1 -15719.268,E2 -15719.268} C_VEL
LIN {X 0,Y 331.801,Z 585.239,A -85,B 0,C 180,E1 -15719.885,E2 -15719.885} C_VEL
LIN {X 0,Y 330.364,Z 598.315,A -85,B 0,C 180,E1 -15720.618,E2 -15720.618} C_VEL
LIN {X 0,Y 328.462,Z 612.799,A -85,B 0,C 180,E1 -15721.689,E2 -15721.689} C_VEL
LIN {X 0,Y 326.282,Z 626.18,A -85,B 0,C 180,E1 -15722.933,E2 -15722.933} C_VEL
LIN {X 0,Y 323.879,Z 639.305,A -85,B 0,C 180,E1 -15724.451,E2 -15724.451} C_VEL
LIN {X 0,Y 321.465,Z 651.286,A -85,B 0,C 180,E1 -15726.143,E2 -15726.143} C_VEL
LIN {X 0,Y 319.286,Z 662.238,A -85,B 0,C 180,E1 -15728.025,E2 -15728.025} C_VEL
LIN {X 0,Y 316.921,Z 672.865,A -85,B 0,C 180,E1 -15730.234,E2 -15730.234} C_VEL
LIN {X 0,Y 315,Z 681.711,A -85,B 0,C 180,E1 -15732.47,E2 -15732.47} C_VEL
LIN {X 0,Y 313.328,Z 690.094,A -85,B 0,C 180,E1 -15735.093,E2 -15735.093} C_VEL
LIN {X 0,Y 312.152,Z 696.613,A -85,B 0,C 180,E1 -15737.649,E2 -15737.649} C_VEL
LIN {X 0,Y 311.333,Z 701.804,A -85,B 0,C 180,E1 -15740.252,E2 -15740.252} C_VEL
LIN {X 0,Y 310.957,Z 704.79,A -85,B 0,C 180,E1 -15742.206,E2 -15742.206} C_VEL
LIN {X 0,Y 310.685,Z 707.728,A -85,B 0,C 180,E1 -15744.808,E2 -15744.808} C_VEL
LIN {X 0,Y 310.647,Z 709.489,A -85,B 0,C 180,E1 -15747.406,E2 -15747.406} C_VEL
LIN {X 0,Y 310.593,Z 710.098,A -85,B 0,C 180,E1 -15750,E2 -15750} C_VEL
LIN {X 0,Y 310.647,Z 709.526,A -85,B 0,C 180,E1 -15752.593,E2 -15752.593} C_VEL
LIN {X 0,Y 310.692,Z 707.815,A -85,B 0,C 180,E1 -15755.191,E2 -15755.191} C_VEL
LIN {X 0,Y 310.971,Z 704.935,A -85,B 0,C 180,E1 -15757.793,E2 -15757.793} C_VEL
LIN {X 0,Y 311.476,Z 700.815,A -85,B 0,C 180,E1 -15760.399,E2 -15760.399} C_VEL
LIN {X 0,Y 312.405,Z 695.346,A -85,B 0,C 180,E1 -15763.001,E2 -15763.001} C_VEL
LIN {X 0,Y 313.665,Z 688.38,A -85,B 0,C 180,E1 -15765.597,E2 -15765.597} C_VEL
LIN {X 0,Y 315.206,Z 680.924,A -85,B 0,C 180,E1 -15767.853,E2 -15767.853} C_VEL
LIN {X 0,Y 317.122,Z 671.941,A -85,B 0,C 180,E1 -15770.091,E2 -15770.091} C_VEL
LIN {X 0,Y 319.371,Z 661.781,A -85,B 0,C 180,E1 -15772.172,E2 -15772.172} C_VEL
LIN {X 0,Y 321.184,Z 652.854,A -85,B 0,C 180,E1 -15773.711,E2 -15773.711} C_VEL
LIN {X 0,Y 321.484,Z 648.549,A -85,B 0,C 180,E1 -15774.432,E2 -15774.432} C_VEL
LIN {X 0,Y 320.319,Z 641.466,A -85,B 0,C 180,E1 -15775.655,E2 -15775.655} C_VEL
LIN {X 0,Y 319.147,Z 634.061,A -85,B 0,C 180,E1 -15776.814,E2 -15776.814} C_VEL
LIN {X 0,Y 319.416,Z 629.216,A -85,B 0,C 180,E1 -15777.422,E2 -15777.422} C_VEL
LIN {X 0,Y 321.708,Z 616.13,A -85,B 0,C 180,E1 -15778.725,E2 -15778.725} C_VEL
LIN {X 0,Y 323.746,Z 602.017,A -85,B 0,C 180,E1 -15779.851,E2 -15779.851} C_VEL
LIN {X 0,Y 325.419,Z 587.797,A -85,B 0,C 180,E1 -15780.724,E2 -15780.724} C_VEL
LIN {X 0,Y 326.853,Z 572.729,A -85,B 0,C 180,E1 -15781.383,E2 -15781.383} C_VEL
LIN {X 0,Y 327.756,Z 557.259,A -85,B 0,C 180,E1 -15781.827,E2 -15781.827} C_VEL
LIN {X 0,Y 331.658,Z 444.395,A -85,B 0,C 180,E1 -15784.266,E2 -15784.266} C_VEL
LIN {X 0,Y 327.805,Z 422.297,A -85,B 0,C 180,E1 -15785.303,E2 -15785.303} C_VEL
LIN {X 0,Y 320.881,Z 407.084,A -85,B 0,C 180,E1 -15786.593,E2 -15786.593} C_VEL
LIN {X 0,Y 315.252,Z 395.734,A -85,B 0,C 180,E1 -15787.713,E2 -15787.713} C_VEL
LIN {X 0,Y 311.414,Z 383.849,A -85,B 0,C 180,E1 -15790.51,E2 -15790.51} C_VEL
LIN {X 0,Y 307.643,Z 373.104,A -85,B 0,C 180,E1 -15793.262,E2 -15793.262} C_VEL
LIN {X 0,Y 305.404,Z 367.29,A -85,B 0,C 180,E1 -15794.917,E2 -15794.917} C_VEL
LIN {X 0,Y 305.412,Z 367.062,A -85,B 0,C 180,E1 -15798.138,E2 -15798.138} C_VEL
LIN {X 0,Y 305.441,Z 367.056,A -85,B 0,C 180,E1 -15801.592,E2 -15801.592} C_VEL
LIN {X 0,Y 305.461,Z 367.049,A -85,B 0,C 180,E1 -15804.886,E2 -15804.886} C_VEL
LIN {X 0,Y 305.441,Z 367.048,A -85,B 0,C 180,E1 -15808.358,E2 -15808.358} C_VEL
LIN {X 0,Y 305.475,Z 367.058,A -85,B 0,C 180,E1 -15811.109,E2 -15811.109} C_VEL
LIN {X 0,Y 305.5,Z 367.046,A -85,B 0,C 180,E1 -15814.081,E2 -15814.081} C_VEL
LIN {X 0,Y 305.473,Z 367.044,A -85,B 0,C 180,E1 -15816.976,E2 -15816.976} C_VEL
LIN {X 0,Y 305.543,Z 367.047,A -85,B 0,C 180,E1 -15821.214,E2 -15821.214} C_VEL
LIN {X 0,Y 305.627,Z 367.036,A -85,B 0,C 180,E1 -15825.348,E2 -15825.348} C_VEL
LIN {X 0,Y 305.625,Z 367.016,A -85,B 0,C 180,E1 -15829.399,E2 -15829.399} C_VEL
LIN {X 0,Y 305.772,Z 367.022,A -85,B 0,C 180,E1 -15832.073,E2 -15832.073} C_VEL
LIN {X 0,Y 305.677,Z 367.009,A -85,B 0,C 180,E1 -15834.723,E2 -15834.723} C_VEL
LIN {X 0,Y 305.954,Z 366.999,A -85,B 0,C 180,E1 -15838.684,E2 -15838.684} C_VEL
LIN {X 0,Y 305.954,Z 366.973,A -85,B 0,C 180,E1 -15841.316,E2 -15841.316} C_VEL
LIN {X 0,Y 305.672,Z 367.031,A -85,B 0,C 180,E1 -15845.277,E2 -15845.277} C_VEL
LIN {X 0,Y 305.752,Z 366.997,A -85,B 0,C 180,E1 -15847.927,E2 -15847.927} C_VEL
LIN {X 0,Y 305.6,Z 367.035,A -85,B 0,C 180,E1 -15851.945,E2 -15851.945} C_VEL
LIN {X 0,Y 305.61,Z 367.024,A -85,B 0,C 180,E1 -15855.015,E2 -15855.015} C_VEL
LIN {X 0,Y 305.543,Z 367.028,A -85,B 0,C 180,E1 -15859.427,E2 -15859.427} C_VEL
LIN {X 0,Y 305.491,Z 367.054,A -85,B 0,C 180,E1 -15863.041,E2 -15863.041} C_VEL
LIN {X 0,Y 305.548,Z 367.04,A -85,B 0,C 180,E1 -15866.227,E2 -15866.227} C_VEL
LIN {X 0,Y 305.495,Z 367.043,A -85,B 0,C 180,E1 -15869.05,E2 -15869.05} C_VEL
LIN {X 0,Y 305.444,Z 367.064,A -85,B 0,C 180,E1 -15871.952,E2 -15871.952} C_VEL
LIN {X 0,Y 305.462,Z 367.048,A -85,B 0,C 180,E1 -15875.113,E2 -15875.113} C_VEL
LIN {X 0,Y 305.439,Z 367.025,A -85,B 0,C 180,E1 -15878.526,E2 -15878.526} C_VEL
LIN {X 0,Y 305.454,Z 367.038,A -85,B 0,C 180,E1 -15882.586,E2 -15882.586} C_VEL
LIN {X 0,Y 305.425,Z 367.024,A -85,B 0,C 180,E1 -15886.345,E2 -15886.345} C_VEL
LIN {X 0,Y 305.465,Z 367.227,A -85,B 0,C 180,E1 -15888.495,E2 -15888.495} C_VEL
LIN {X 0,Y 305.75,Z 368.437,A -85,B 0,C 180,E1 -15888.819,E2 -15888.819} C_VEL
LIN {X 0,Y 307.85,Z 372.313,A -85,B 0,C 180,E1 -15889.565,E2 -15889.565} C_VEL
LIN {X 0,Y 315.343,Z 392.445,A -85,B 0,C 180,E1 -15892.565,E2 -15892.565} C_VEL
LIN {X 0,Y 326.403,Z 416.818,A -85,B 0,C 180,E1 -15894.691,E2 -15894.691} C_VEL
LIN {X 0,Y 328.377,Z 421.825,A -85,B 0,C 180,E1 -15895.067,E2 -15895.067} C_VEL
LIN {X 0,Y 331.088,Z 440.61,A -85,B 0,C 180,E1 -15895.879,E2 -15895.879} C_VEL
LIN {X 0,Y 326.986,Z 561.183,A -85,B 0,C 180,E1 -15898.496,E2 -15898.496} C_VEL
LIN {X 0,Y 325.933,Z 577.042,A -85,B 0,C 180,E1 -15899.015,E2 -15899.015} C_VEL
LIN {X 0,Y 324.411,Z 592.108,A -85,B 0,C 180,E1 -15899.756,E2 -15899.756} C_VEL
LIN {X 0,Y 322.698,Z 605.503,A -85,B 0,C 180,E1 -15900.645,E2 -15900.645} C_VEL
LIN {X 0,Y 320.551,Z 619.851,A -85,B 0,C 180,E1 -15901.876,E2 -15901.876} C_VEL
LIN {X 0,Y 318.205,Z 632.779,A -85,B 0,C 180,E1 -15903.256,E2 -15903.256} C_VEL
LIN {X 0,Y 315.894,Z 644.689,A -85,B 0,C 180,E1 -15904.818,E2 -15904.818} C_VEL
LIN {X 0,Y 313.641,Z 655.408,A -85,B 0,C 180,E1 -15906.507,E2 -15906.507} C_VEL
LIN {X 0,Y 311.449,Z 665.82,A -85,B 0,C 180,E1 -15908.489,E2 -15908.489} C_VEL
LIN {X 0,Y 309.151,Z 675.692,A -85,B 0,C 180,E1 -15910.754,E2 -15910.754} C_VEL
LIN {X 0,Y 307.336,Z 683.876,A -85,B 0,C 180,E1 -15913.049,E2 -15913.049} C_VEL
LIN {X 0,Y 305.988,Z 690.642,A -85,B 0,C 180,E1 -15915.366,E2 -15915.366} C_VEL
LIN {X 0,Y 304.808,Z 696.908,A -85,B 0,C 180,E1 -15918.023,E2 -15918.023} C_VEL
LIN {X 0,Y 304.156,Z 701.74,A -85,B 0,C 180,E1 -15920.692,E2 -15920.692} C_VEL
LIN {X 0,Y 303.724,Z 705.272,A -85,B 0,C 180,E1 -15923.356,E2 -15923.356} C_VEL
LIN {X 0,Y 303.581,Z 707.595,A -85,B 0,C 180,E1 -15926.018,E2 -15926.018} C_VEL
LIN {X 0,Y 303.536,Z 708.762,A -85,B 0,C 180,E1 -15928.673,E2 -15928.673} C_VEL
LIN {X 0,Y 303.537,Z 708.761,A -85,B 0,C 180,E1 -15931.327,E2 -15931.327} C_VEL
LIN {X 0,Y 303.582,Z 707.587,A -85,B 0,C 180,E1 -15933.983,E2 -15933.983} C_VEL
LIN {X 0,Y 303.724,Z 705.255,A -85,B 0,C 180,E1 -15936.644,E2 -15936.644} C_VEL
LIN {X 0,Y 304.156,Z 701.707,A -85,B 0,C 180,E1 -15939.308,E2 -15939.308} C_VEL
LIN {X 0,Y 304.815,Z 696.861,A -85,B 0,C 180,E1 -15941.977,E2 -15941.977} C_VEL
LIN {X 0,Y 305.988,Z 690.591,A -85,B 0,C 180,E1 -15944.635,E2 -15944.635} C_VEL
LIN {X 0,Y 307.382,Z 683.813,A -85,B 0,C 180,E1 -15946.949,E2 -15946.949} C_VEL
LIN {X 0,Y 309.15,Z 675.611,A -85,B 0,C 180,E1 -15949.247,E2 -15949.247} C_VEL
LIN {X 0,Y 311.428,Z 665.719,A -85,B 0,C 180,E1 -15951.513,E2 -15951.513} C_VEL
LIN {X 0,Y 314.954,Z 651.21,A -85,B 0,C 180,E1 -15954.382,E2 -15954.382} C_VEL
LIN {X 0,Y 318.034,Z 640.622,A -85,B 0,C 180,E1 -15956.23,E2 -15956.23} C_VEL
LIN {X 0,Y 321.459,Z 628.231,A -85,B 0,C 180,E1 -15958.038,E2 -15958.038} C_VEL
LIN {X 0,Y 324.994,Z 614.786,A -85,B 0,C 180,E1 -15959.648,E2 -15959.648} C_VEL
LIN {X 0,Y 328.464,Z 600.638,A -85,B 0,C 180,E1 -15961.023,E2 -15961.023} C_VEL
LIN {X 0,Y 331.921,Z 585.01,A -85,B 0,C 180,E1 -15962.23,E2 -15962.23} C_VEL
LIN {X 0,Y 334.95,Z 569.266,A -85,B 0,C 180,E1 -15963.151,E2 -15963.151} C_VEL
LIN {X 0,Y 337.471,Z 553.241,A -85,B 0,C 180,E1 -15963.854,E2 -15963.854} C_VEL
LIN {X 0,Y 347.11,Z 482.201,A -85,B 0,C 180,E1 -15966.474,E2 -15966.474} C_VEL
LIN {X 0,Y 352.511,Z 447.115,A -85,B 0,C 180,E1 -15967.795,E2 -15967.795} C_VEL
LIN {X 0,Y 350.599,Z 442.205,A -85,B 0,C 180,E1 -15969.027,E2 -15969.027} C_VEL
LIN {X 0,Y 348.256,Z 436.995,A -85,B 0,C 180,E1 -15970.814,E2 -15970.814} C_VEL
LIN {X 0,Y 346.186,Z 433.061,A -85,B 0,C 180,E1 -15973.043,E2 -15973.043} C_VEL
LIN {X 0,Y 345.218,Z 431.724,A -85,B 0,C 180,E1 -15974.779,E2 -15974.779} C_VEL
LIN {X 0,Y 344.951,Z 431.574,A -85,B 0,C 180,E1 -15977.178,E2 -15977.178} C_VEL
LIN {X 0,Y 345.774,Z 432.912,A -85,B 0,C 180,E1 -15979.277,E2 -15979.277} C_VEL
LIN {X 0,Y 347.605,Z 436.967,A -85,B 0,C 180,E1 -15981.602,E2 -15981.602} C_VEL
LIN {X 0,Y 349.782,Z 442.345,A -85,B 0,C 180,E1 -15983.485,E2 -15983.485} C_VEL
LIN {X 0,Y 351.673,Z 447.73,A -85,B 0,C 180,E1 -15984.844,E2 -15984.844} C_VEL
LIN {X 0,Y 351.68,Z 451.381,A -85,B 0,C 180,E1 -15985.207,E2 -15985.207} C_VEL
LIN {X 0,Y 338.612,Z 535.422,A -85,B 0,C 180,E1 -15988.569,E2 -15988.569} C_VEL
LIN {X 0,Y 335.885,Z 553.84,A -85,B 0,C 180,E1 -15989.379,E2 -15989.379} C_VEL
LIN {X 0,Y 332.939,Z 570.04,A -85,B 0,C 180,E1 -15990.359,E2 -15990.359} C_VEL
LIN {X 0,Y 329.586,Z 586.28,A -85,B 0,C 180,E1 -15991.676,E2 -15991.676} C_VEL
LIN {X 0,Y 326.209,Z 600.247,A -85,B 0,C 180,E1 -15993.1,E2 -15993.1} C_VEL
LIN {X 0,Y 322.835,Z 613,A -85,B 0,C 180,E1 -15994.708,E2 -15994.708} C_VEL
LIN {X 0,Y 319.848,Z 623.722,A -85,B 0,C 180,E1 -15996.359,E2 -15996.359} C_VEL
LIN {X 0,Y 316.956,Z 633.64,A -85,B 0,C 180,E1 -15998.198,E2 -15998.198} C_VEL
LIN {X 0,Y 313.917,Z 643.364,A -85,B 0,C 180,E1 -16000.378,E2 -16000.378} C_VEL
LIN {X 0,Y 311.277,Z 651.348,A -85,B 0,C 180,E1 -16002.593,E2 -16002.593} C_VEL
LIN {X 0,Y 309.157,Z 657.826,A -85,B 0,C 180,E1 -16004.845,E2 -16004.845} C_VEL
LIN {X 0,Y 307.283,Z 663.588,A -85,B 0,C 180,E1 -16007.451,E2 -16007.451} C_VEL
LIN {X 0,Y 306.267,Z 666.891,A -85,B 0,C 180,E1 -16009.422,E2 -16009.422} C_VEL
LIN {X 0,Y 305.064,Z 670.022,A -85,B 0,C 180,E1 -16012.055,E2 -16012.055} C_VEL
LIN {X 0,Y 304.302,Z 671.699,A -85,B 0,C 180,E1 -16014.699,E2 -16014.699} C_VEL
LIN {X 0,Y 303.996,Z 671.944,A -85,B 0,C 180,E1 -16017.35,E2 -16017.35} C_VEL
LIN {X 0,Y 303.759,Z 670.768,A -85,B 0,C 180,E1 -16020,E2 -16020} C_VEL
LIN {X 0,Y 303.776,Z 668.136,A -85,B 0,C 180,E1 -16022.652,E2 -16022.652} C_VEL
LIN {X 0,Y 303.882,Z 665.19,A -85,B 0,C 180,E1 -16024.643,E2 -16024.643} C_VEL
LIN {X 0,Y 304.172,Z 659.776,A -85,B 0,C 180,E1 -16027.301,E2 -16027.301} C_VEL
LIN {X 0,Y 304.575,Z 653.579,A -85,B 0,C 180,E1 -16029.631,E2 -16029.631} C_VEL
LIN {X 0,Y 305.22,Z 645.819,A -85,B 0,C 180,E1 -16031.96,E2 -16031.96} C_VEL
LIN {X 0,Y 306.124,Z 637.741,A -85,B 0,C 180,E1 -16033.949,E2 -16033.949} C_VEL
LIN {X 0,Y 307.131,Z 627.545,A -85,B 0,C 180,E1 -16036.038,E2 -16036.038} C_VEL
LIN {X 0,Y 308.375,Z 616.416,A -85,B 0,C 180,E1 -16037.919,E2 -16037.919} C_VEL
LIN {X 0,Y 309.577,Z 604.641,A -85,B 0,C 180,E1 -16039.564,E2 -16039.564} C_VEL
LIN {X 0,Y 311.018,Z 591.929,A -85,B 0,C 180,E1 -16041.022,E2 -16041.022} C_VEL
LIN {X 0,Y 312.332,Z 578.043,A -85,B 0,C 180,E1 -16042.316,E2 -16042.316} C_VEL
LIN {X 0,Y 313.511,Z 562.63,A -85,B 0,C 180,E1 -16043.447,E2 -16043.447} C_VEL
LIN {X 0,Y 314.544,Z 546.99,A -85,B 0,C 180,E1 -16044.284,E2 -16044.284} C_VEL
LIN {X 0,Y 315.525,Z 526.282,A -85,B 0,C 180,E1 -16045.037,E2 -16045.037} C_VEL
LIN {X 0,Y 319.746,Z 437.478,A -85,B 0,C 180,E1 -16047.931,E2 -16047.931} C_VEL
LIN {X 0,Y 314.691,Z 403.56,A -85,B 0,C 180,E1 -16049.492,E2 -16049.492} C_VEL
LIN {X 0,Y 312.689,Z 397.96,A -85,B 0,C 180,E1 -16049.89,E2 -16049.89} C_VEL
LIN {X 0,Y 309.62,Z 384.143,A -85,B 0,C 180,E1 -16053.397,E2 -16053.397} C_VEL
LIN {X 0,Y 306.67,Z 371.973,A -85,B 0,C 180,E1 -16056.668,E2 -16056.668} C_VEL
LIN {X 0,Y 305.446,Z 367.182,A -85,B 0,C 180,E1 -16058.084,E2 -16058.084} C_VEL
